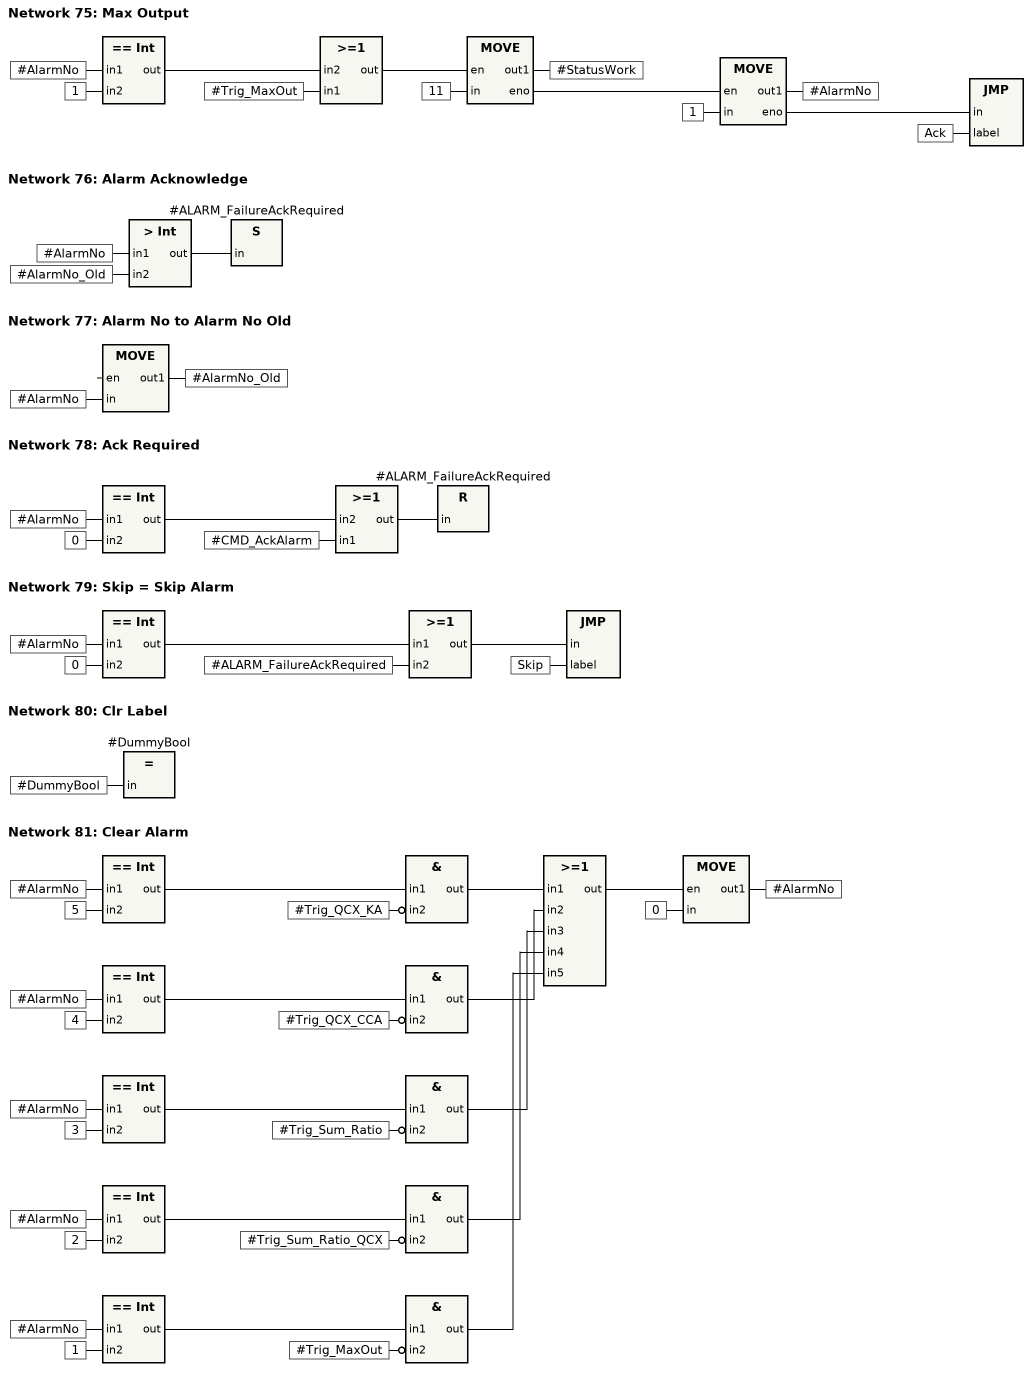
   // ENO of a box is taken as its EN; it also drops when the box reports an error
   #_w1 := (#AlarmNo = 1) OR #Trig_MaxOut;
   IF #_w1 THEN
       #StatusWork := 11;
       #AlarmNo := 1;
       GOTO Ack;
   END_IF;
END_REGION

REGION Network 76: Alarm Acknowledge
   Ack:
   IF #AlarmNo > #AlarmNo_Old THEN #ALARM_FailureAckRequired := TRUE; END_IF;
END_REGION

REGION Network 77: Alarm No to Alarm No Old
   #AlarmNo_Old := #AlarmNo;
END_REGION

REGION Network 78: Ack Required
   IF (#AlarmNo = 0) OR #CMD_AckAlarm THEN #ALARM_FailureAckRequired := FALSE; END_IF;
END_REGION

REGION Network 79: Skip = Skip Alarm
   IF (#AlarmNo = 0) OR #ALARM_FailureAckRequired THEN GOTO Skip; END_IF;
END_REGION

REGION Network 80: Clr Label
   Clr:
   #DummyBool := #DummyBool;
END_REGION

REGION Network 81: Clear Alarm
   IF ((#AlarmNo = 5) AND NOT #Trig_QCX_KA) OR ((#AlarmNo = 4) AND NOT #Trig_QCX_CCA) OR ((#AlarmNo = 3) AND NOT #Trig_Sum_Ratio) OR ((#AlarmNo = 2) AND NOT #Trig_Sum_Ratio_QCX) OR ((#AlarmNo = 1) AND NOT #Trig_MaxOut) THEN
       #AlarmNo := 0;
   END_IF;
END_REGION

REGION Network 82: Clear Alarm No Old
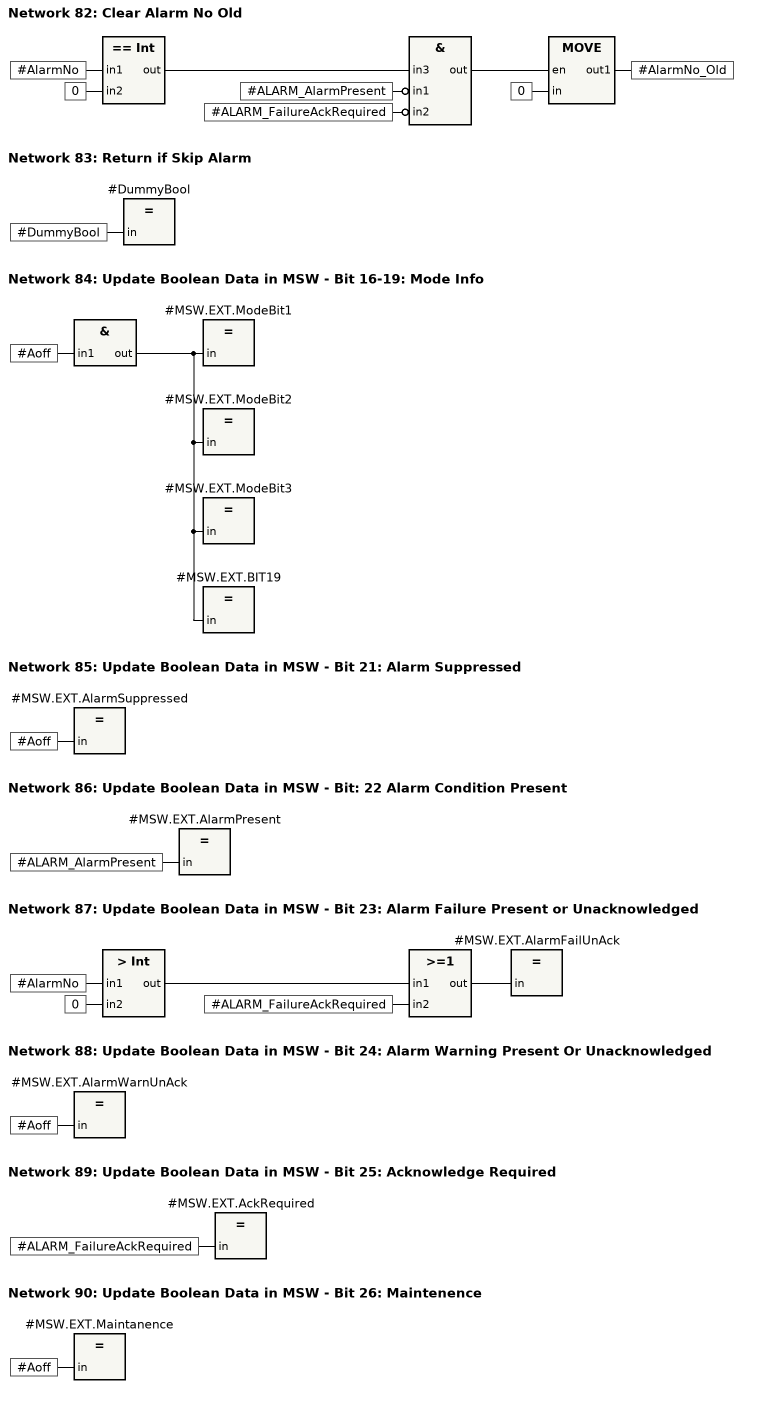
   IF (#AlarmNo = 0) AND NOT #ALARM_AlarmPresent AND NOT #ALARM_FailureAckRequired THEN
       #AlarmNo_Old := 0;
   END_IF;
END_REGION

REGION Network 83: Return if Skip Alarm
   Skip:
   #DummyBool := #DummyBool;
END_REGION

REGION Network 84: Update Boolean Data in MSW - Bit 16-19: Mode Info
   // 0 = Auto
   // 1= Single Start
   // 2 = Manual
   // 3= Local
   // 4= Test Mode
   #MSW.EXT.ModeBit1 := #Aoff;
   #MSW.EXT.ModeBit2 := #Aoff;
   #MSW.EXT.ModeBit3 := #Aoff;
   #MSW.EXT.BIT19 := #Aoff;
END_REGION

REGION Network 85: Update Boolean Data in MSW - Bit 21: Alarm Suppressed
   #MSW.EXT.AlarmSuppressed := #Aoff;
END_REGION

REGION Network 86: Update Boolean Data in MSW - Bit: 22 Alarm Condition Present
   #MSW.EXT.AlarmPresent := #ALARM_AlarmPresent;
END_REGION

REGION Network 87: Update Boolean Data in MSW - Bit 23: Alarm Failure Present or Unacknowledged
   #MSW.EXT.AlarmFailUnAck := (#AlarmNo > 0) OR #ALARM_FailureAckRequired;
END_REGION

REGION Network 88: Update Boolean Data in MSW - Bit 24: Alarm Warning Present Or Unacknowledged
   #MSW.EXT.AlarmWarnUnAck := #Aoff;
END_REGION

REGION Network 89: Update Boolean Data in MSW - Bit 25: Acknowledge Required
   #MSW.EXT.AckRequired := #ALARM_FailureAckRequired;
END_REGION

REGION Network 90: Update Boolean Data in MSW - Bit 26: Maintenence
   #MSW.EXT.Maintanence := #Aoff;
END_REGION

REGION Network 91: Update Boolean Data in MSW - Bit 27: Operation
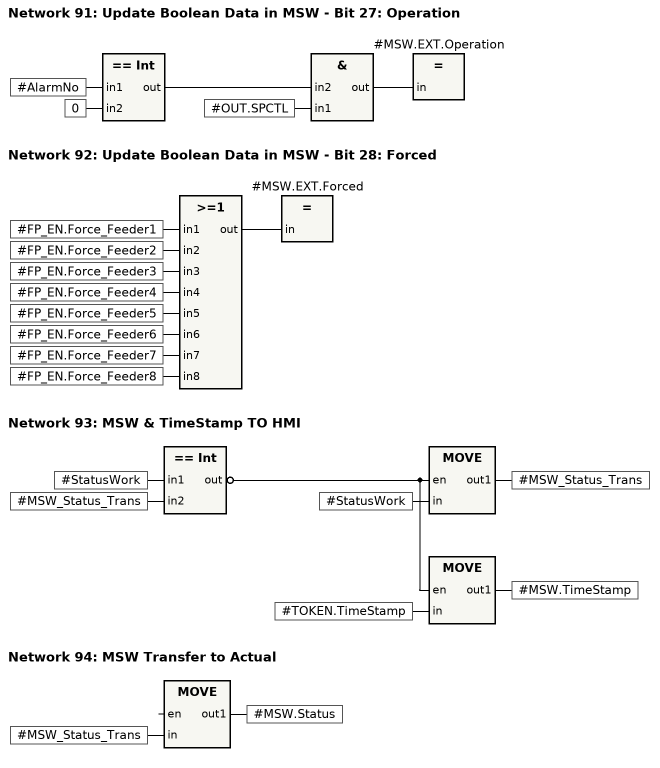
   #MSW.EXT.Operation := (#AlarmNo = 0) AND #OUT.SPCTL;
END_REGION

REGION Network 92: Update Boolean Data in MSW - Bit 28: Forced
   #MSW.EXT.Forced := #FP_EN.Force_Feeder1 OR #FP_EN.Force_Feeder2 OR #FP_EN.Force_Feeder3 OR #FP_EN.Force_Feeder4 OR #FP_EN.Force_Feeder5 OR #FP_EN.Force_Feeder6 OR #FP_EN.Force_Feeder7 OR #FP_EN.Force_Feeder8;
END_REGION

REGION Network 93: MSW & TimeStamp TO HMI
   #_w1 := NOT (#StatusWork = #MSW_Status_Trans);
   IF #_w1 THEN
       #MSW_Status_Trans := #StatusWork;
       #MSW.TimeStamp := #TOKEN.TimeStamp;
   END_IF;
END_REGION

REGION Network 94: MSW Transfer to Actual
   #MSW.Status := #MSW_Status_Trans;
END_REGION

REGION Network 95: Write STAT to OUT
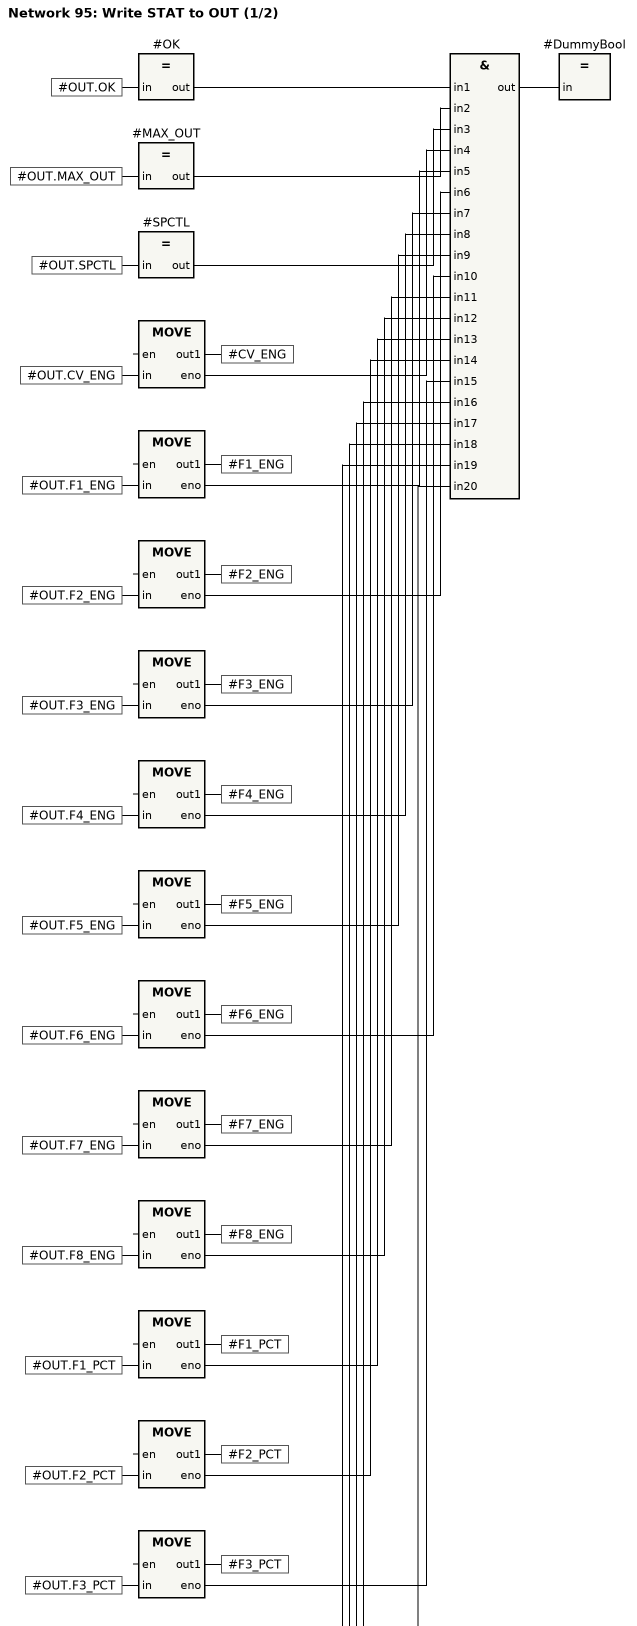
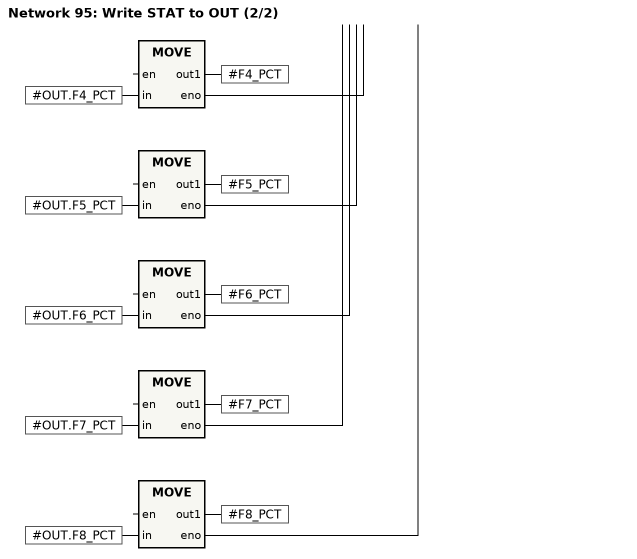
   #OK := #OUT.OK;
   #MAX_OUT := #OUT.MAX_OUT;
   #SPCTL := #OUT.SPCTL;
   #CV_ENG := #OUT.CV_ENG;
   #F1_ENG := #OUT.F1_ENG;
   #F2_ENG := #OUT.F2_ENG;
   #F3_ENG := #OUT.F3_ENG;
   #F4_ENG := #OUT.F4_ENG;
   #F5_ENG := #OUT.F5_ENG;
   #F6_ENG := #OUT.F6_ENG;
   #F7_ENG := #OUT.F7_ENG;
   #F8_ENG := #OUT.F8_ENG;
   #F1_PCT := #OUT.F1_PCT;
   #F2_PCT := #OUT.F2_PCT;
   #F3_PCT := #OUT.F3_PCT;
   #F4_PCT := #OUT.F4_PCT;
   #F5_PCT := #OUT.F5_PCT;
   #F6_PCT := #OUT.F6_PCT;
   #F7_PCT := #OUT.F7_PCT;
   #F8_PCT := #OUT.F8_PCT;
   #DummyBool := #OUT.OK AND #OUT.MAX_OUT AND #OUT.SPCTL;
END_REGION
END_FUNCTION_BLOCK

FUNCTION_BLOCK "ACESYS_SEQUENCE"   // FB231, FBD
TITLE = ACESYS V8.0 - Build 003 - SEQUENCE
{ S7_Optimized_Access := 'FALSE' }
AUTHOR : FLSmidth
FAMILY : ACESYS
NAME : SEQ
VERSION : 8.0
   VAR_INPUT
      TRANS_01 : Bool := TRUE;   // Transition 01
      TRANS_02 : Bool := TRUE;   // Transition 02
      TRANS_03 : Bool := TRUE;   // Transition 03
      TRANS_04 : Bool := TRUE;   // Transition 04
      TRANS_05 : Bool := TRUE;   // Transition 05
      TRANS_06 : Bool := TRUE;   // Transition 06
      TRANS_07 : Bool := TRUE;   // Transition 07
      TRANS_08 : Bool := TRUE;   // Transition 08
      TRANS_09 : Bool := TRUE;   // Transition 09
      TRANS_10 : Bool := TRUE;   // Transition 10
      TRANS_11 : Bool := TRUE;   // Transition 11
      TRANS_12 : Bool := TRUE;   // Transition 12
      TRANS_13 : Bool := TRUE;   // Transition 13
      TRANS_14 : Bool := TRUE;   // Transition 14
      TRANS_15 : Bool := TRUE;   // Transition 15
      TRANS_16 : Bool := TRUE;   // Transition 16
      RESET : Bool;   // Reset to Step 1
      SINGLE_STEP : Bool;   // Goto Next Step
      GOTO_STEP : Bool;   // Goto step Request
      GOTO_NO : Int;   // Goto step Number
   END_VAR
   VAR_OUTPUT
      OUT_01 : Bool;   // Output 01
      OUT_02 : Bool;   // Output 02
      OUT_03 : Bool;   // Output 03
      OUT_04 : Bool;   // Output 04
      OUT_05 : Bool;   // Output 05
      OUT_06 : Bool;   // Output 06
      OUT_07 : Bool;   // Output 07
      OUT_08 : Bool;   // Output 08
      OUT_09 : Bool;   // Output 09
      OUT_10 : Bool;   // Output 10
      OUT_11 : Bool;   // Output 11
      OUT_12 : Bool;   // Output 12
      OUT_13 : Bool;   // Output 13
      OUT_14 : Bool;   // Output 14
      OUT_15 : Bool;   // Output 15
      OUT_16 : Bool;   // Output 16
      OK : Bool := TRUE;   // Unit OK (1=no alarms)
      MAX_TIME : Bool;   // Max Step time exceeded
      ACT_STEP : Int;   // Actual Step
      MSW : "ACESYS_HMI_STAT_32T";
   END_VAR
   VAR_IN_OUT
      TOKEN : "ACESYS_TOKEN";
   END_VAR
   VAR
      BlockInfo : Struct
         Ace_Version : Int;   // Acesys Block Version Number
         Ace_BuildNo : Int;   // Acesys Block Build Number
         DB_Number : Int;   // Block Instance DB Number
      END_STRUCT;
      FP_CMD : Struct   // Faceplate Commands
         Spare_08 : Bool;
         Spare_09 : Bool;
         Spare_10 : Bool;
         Spare_11 : Bool;
         Spare_12 : Bool;
         Spare_13 : Bool;
         Spare_14 : Bool;
         AckAlarm : Bool;   // Alarm Acknowledge
         GotoStep1 : Bool;   // FacePlateCmd (bit 0): Reset Sequence to Step 1
         GotoNext : Bool;   // FacePlateCmd (bit 1): Goto Next STep
         Spare_02 : Bool;
         Spare_03 : Bool;
         Spare_04 : Bool;
         Spare_05 : Bool;
         Spare_06 : Bool;
         Spare_07 : Bool;
      END_STRUCT;
      FP_SEL : Struct
         Alarm_Type_1 : Bool;   // No Alarm
         Alarm_Type_2 : Bool;   // Alarm Warming
         Alarm_Type_3 : Bool;   // Alarm Failure
         Alarm_Type_4 : Bool;   // Spare (not Used)
         Alarm_Action_1 : Bool;   // No Action
         Alarm_Action_2 : Bool;   // Continue to next Step
         Alarm_Action_3 : Bool;   // Reset to Step 1
         Alarm_Action_4 : Bool;   // Spare (Not Used)
         Retentive_Timer : Bool;
      END_STRUCT;
      FP_PARM : Struct
         MATRIX : Array[1..16] of Word;   // Output Matrix
         Min_Time_Pre : Array[1..16] of DInt;   // Minumum Step Time
         Max_Time_Pre : Array[1..16] of DInt;   // Maximum Step Time
         Min_Time_Acc : DInt;   // Min Step time Actual
         Max_Time_Acc : DInt;   // Max Step time Actual
         Min_Time_SP : DInt;   // Min Step time Setpoint
         Max_Time_SP : DInt;   // Max Step time Setpoint
         NoOfOutputs : Int := 16;   // Number Outputs to be displayed on faceplate
         NoOfSteps : Int := 16;   // Number of Steps to be displayed on faceplate
         Min_Timer_EN : Bool;   // Minimum Step Timer Enabled
         Min_Timer_DN : Bool;   // Minimum Step Timer Elapsed
         Max_Timer_EN : Bool;   // Maximum Step Timer Enabled
         Max_Timer_DN : Bool;   // Maximum Step Time Elapsed
         Trans_Act : Bool;   // Active Transition
      END_STRUCT;
      FP_DIM : Struct
         GotoStep1 : Bool;
         GotoNext : Bool;
      END_STRUCT;
      FP_SHOW : Struct
         GotoStep1 : Bool;
         GotoNext : Bool;
      END_STRUCT;
      ONS : Struct
         Alarm_Type_1 : Bool;
         Alarm_Type_2 : Bool;
         Alarm_Type_3 : Bool;
         Alarm_Type_4 : Bool;
         Alarm_Action_1 : Bool;
         Alarm_Action_2 : Bool;
         Alarm_Action_3 : Bool;
         Alarm_Action_4 : Bool;
         Goto_Step : Bool;
         SingleStep : Bool;
         Reset : Bool;
         Acknowledge : Bool;
      END_STRUCT;
      Work_Step : Int;
      Old_Step : Int;
      StatusWork : Int;
      AlarmNo : Int;
      AlarmNo_Old : Int;
      TimerMin_SP : DInt;
      TimerMin_ACC : DInt;
      TimerMax_SP : DInt;
      TimerMax_ACC : DInt;
      Reset_Timer : Bool;
      ALARM_AlarmPresent : Bool;
      ALARM_WarnPresent : Bool;
      ALARM_FailureAckRequired : Bool;
      ALARM_Warn_Ack_Required : Bool;
      CMD_Acknowledge : Bool;
      Min_Timer : TONR_TIME;
      Max_Timer : TONR_TIME;
      MSW_Status_Trans : Int;
      OUT : Struct
         OUT_01 : Bool;
         OUT_02 : Bool;
         OUT_03 : Bool;
         OUT_04 : Bool;
         OUT_05 : Bool;
         OUT_06 : Bool;
         OUT_07 : Bool;
         OUT_08 : Bool;
         OUT_09 : Bool;
         OUT_10 : Bool;
         OUT_11 : Bool;
         OUT_12 : Bool;
         OUT_13 : Bool;
         OUT_14 : Bool;
         OUT_15 : Bool;
         OUT_16 : Bool;
         OK : Bool;
         MAX_TIME : Bool;
      END_STRUCT;
      Min_Timer_Q : Bool;
      Max_Timer_Q : Bool;
   END_VAR
   VAR_TEMP
      Aon : Bool;
      Aoff : Bool;
      DummyBool : Bool;
      Work_Matrix : Word;
      Work_Matrix_B AT Work_Matrix : Array[0..15] of Bool;
   END_VAR
   VAR_TEMP   // added for the SCL form of the ladder/FBD networks
      _w1 : Bool;
      _w2 : Bool;
      _w3 : Bool;
      _w4 : Bool;
      _w5 : Bool;
      _w6 : Bool;
      _w7 : Bool;
      _w8 : Bool;
      _w9 : Bool;
      _w10 : Bool;
      _w11 : Bool;
      _w12 : Bool;
      _w13 : Bool;
      _w14 : Bool;
      _w15 : Bool;
      _w16 : Bool;
   END_VAR
BEGIN

REGION Network 1
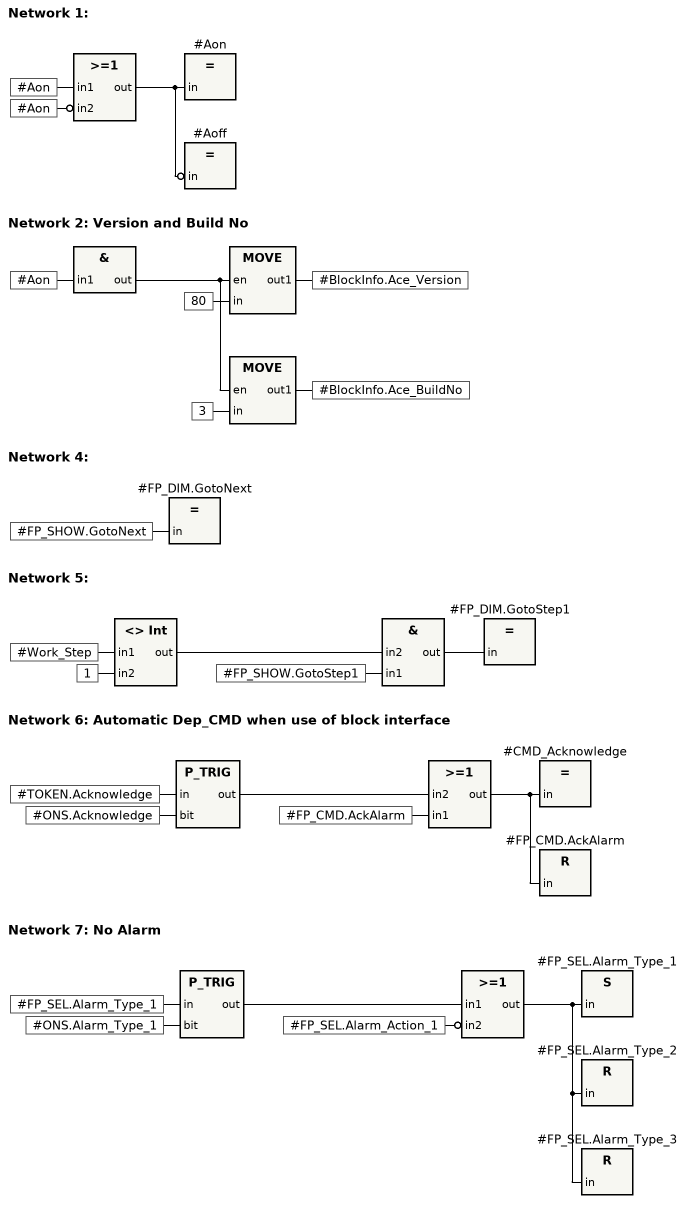
   #Aon := #Aon OR NOT #Aon;
   #Aoff := NOT #Aon;
END_REGION

REGION Network 2: Version and Build No
   IF #Aon THEN
       #BlockInfo.Ace_Version := 80;
       #BlockInfo.Ace_BuildNo := 3;
   END_IF;
END_REGION

REGION Network 3 (STL): Instance DB Number to Faceplate
         L     DINO;
         T     #BlockInfo.DB_Number;
END_REGION

REGION Network 4
   #FP_DIM.GotoNext := #FP_SHOW.GotoNext;
END_REGION

REGION Network 5
   #FP_DIM.GotoStep1 := (#Work_Step <> 1) AND #FP_SHOW.GotoStep1;
END_REGION

REGION Network 6: Automatic Dep_CMD when use of block interface
   #_w1 := #TOKEN.Acknowledge AND NOT #ONS.Acknowledge;   // rising edge
   #ONS.Acknowledge := #TOKEN.Acknowledge;
   #CMD_Acknowledge := #_w1 OR #FP_CMD.AckAlarm;
   IF #CMD_Acknowledge THEN #FP_CMD.AckAlarm := FALSE; END_IF;
END_REGION

REGION Network 7: No Alarm
   // Alarm Type:
   // 
   // 1 = No Alarm
   // 2 = Alarm Warning
   // 3 = Alarm Failure
   #_w1 := #FP_SEL.Alarm_Type_1 AND NOT #ONS.Alarm_Type_1;   // rising edge
   #ONS.Alarm_Type_1 := #FP_SEL.Alarm_Type_1;
   IF #_w1 OR NOT #FP_SEL.Alarm_Action_1 THEN
       #FP_SEL.Alarm_Type_1 := TRUE;
       #FP_SEL.Alarm_Type_2 := FALSE;
       #FP_SEL.Alarm_Type_3 := FALSE;
   END_IF;
END_REGION

REGION Network 8: No Alarm
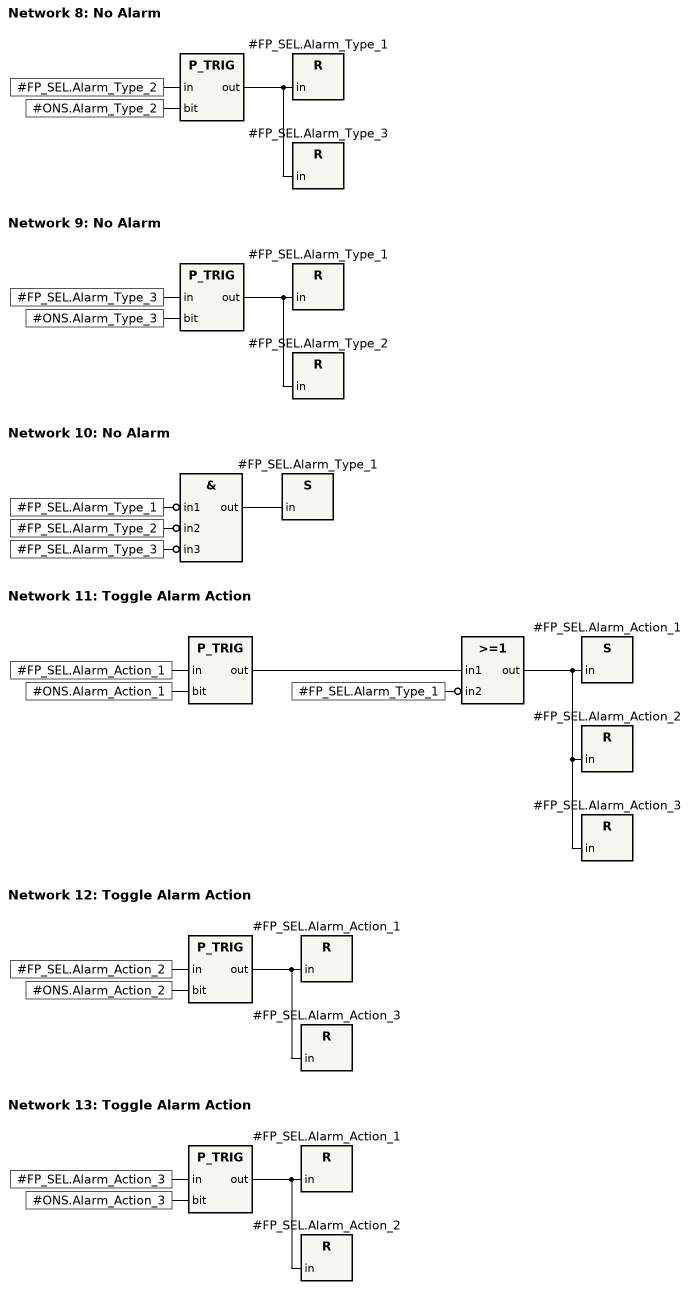
   #_w1 := #FP_SEL.Alarm_Type_2 AND NOT #ONS.Alarm_Type_2;   // rising edge
   #ONS.Alarm_Type_2 := #FP_SEL.Alarm_Type_2;
   IF #_w1 THEN
       #FP_SEL.Alarm_Type_1 := FALSE;
       #FP_SEL.Alarm_Type_3 := FALSE;
   END_IF;
END_REGION

REGION Network 9: No Alarm
   #_w1 := #FP_SEL.Alarm_Type_3 AND NOT #ONS.Alarm_Type_3;   // rising edge
   #ONS.Alarm_Type_3 := #FP_SEL.Alarm_Type_3;
   IF #_w1 THEN
       #FP_SEL.Alarm_Type_1 := FALSE;
       #FP_SEL.Alarm_Type_2 := FALSE;
   END_IF;
END_REGION

REGION Network 10: No Alarm
   IF NOT #FP_SEL.Alarm_Type_1 AND NOT #FP_SEL.Alarm_Type_2 AND NOT #FP_SEL.Alarm_Type_3 THEN
       #FP_SEL.Alarm_Type_1 := TRUE;
   END_IF;
END_REGION

REGION Network 11: Toggle Alarm Action
   // Alarm Action:
   // 
   // 1 = No Action
   // 2 = Continue to Next Step
   // 3 = Reset to Step 1
   // 4 = Stay in current step until Alarm Acknowledged
   #_w1 := #FP_SEL.Alarm_Action_1 AND NOT #ONS.Alarm_Action_1;   // rising edge
   #ONS.Alarm_Action_1 := #FP_SEL.Alarm_Action_1;
   IF #_w1 OR NOT #FP_SEL.Alarm_Type_1 THEN
       #FP_SEL.Alarm_Action_1 := TRUE;
       #FP_SEL.Alarm_Action_2 := FALSE;
       #FP_SEL.Alarm_Action_3 := FALSE;
   END_IF;
END_REGION

REGION Network 12: Toggle Alarm Action
   #_w1 := #FP_SEL.Alarm_Action_2 AND NOT #ONS.Alarm_Action_2;   // rising edge
   #ONS.Alarm_Action_2 := #FP_SEL.Alarm_Action_2;
   IF #_w1 THEN
       #FP_SEL.Alarm_Action_1 := FALSE;
       #FP_SEL.Alarm_Action_3 := FALSE;
   END_IF;
END_REGION

REGION Network 13: Toggle Alarm Action
   #_w1 := #FP_SEL.Alarm_Action_3 AND NOT #ONS.Alarm_Action_3;   // rising edge
   #ONS.Alarm_Action_3 := #FP_SEL.Alarm_Action_3;
   IF #_w1 THEN
       #FP_SEL.Alarm_Action_1 := FALSE;
       #FP_SEL.Alarm_Action_2 := FALSE;
   END_IF;
END_REGION

REGION Network 14: No Action
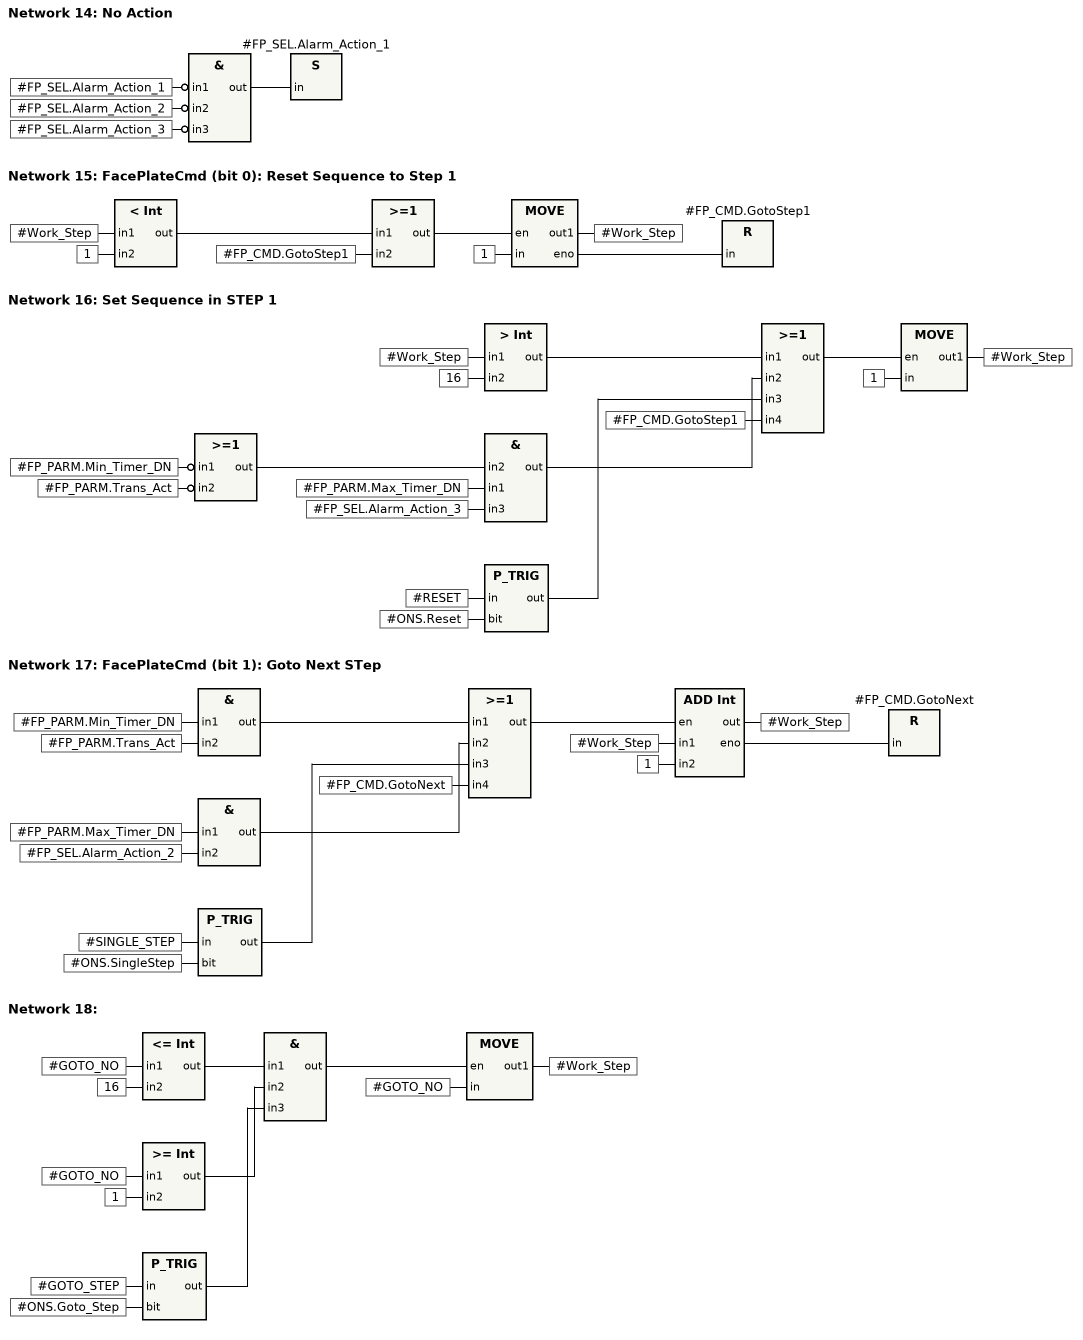
   IF NOT #FP_SEL.Alarm_Action_1 AND NOT #FP_SEL.Alarm_Action_2 AND NOT #FP_SEL.Alarm_Action_3 THEN
       #FP_SEL.Alarm_Action_1 := TRUE;
   END_IF;
END_REGION

REGION Network 15: FacePlateCmd (bit 0): Reset Sequence to Step 1
   // ENO of a box is taken as its EN; it also drops when the box reports an error
   #_w1 := (#Work_Step < 1) OR #FP_CMD.GotoStep1;
   IF #_w1 THEN
       #Work_Step := 1;
       #FP_CMD.GotoStep1 := FALSE;
   END_IF;
END_REGION

REGION Network 16: Set Sequence in STEP 1
   #_w1 := #RESET AND NOT #ONS.Reset;   // rising edge
   #ONS.Reset := #RESET;
   IF (#Work_Step > 16) OR ((NOT #FP_PARM.Min_Timer_DN OR NOT #FP_PARM.Trans_Act) AND #FP_PARM.Max_Timer_DN AND #FP_SEL.Alarm_Action_3) OR #_w1 OR #FP_CMD.GotoStep1 THEN
       #Work_Step := 1;
   END_IF;
END_REGION

REGION Network 17: FacePlateCmd (bit 1): Goto Next STep
   // ENO of a box is taken as its EN; it also drops when the box reports an error
   #_w1 := #SINGLE_STEP AND NOT #ONS.SingleStep;   // rising edge
   #ONS.SingleStep := #SINGLE_STEP;
   IF (#FP_PARM.Min_Timer_DN AND #FP_PARM.Trans_Act) OR (#FP_PARM.Max_Timer_DN AND #FP_SEL.Alarm_Action_2) OR #_w1 OR #FP_CMD.GotoNext THEN
       #Work_Step := #Work_Step + 1;
       #FP_CMD.GotoNext := FALSE;
   END_IF;
END_REGION

REGION Network 18
   #_w1 := #GOTO_STEP AND NOT #ONS.Goto_Step;   // rising edge
   #ONS.Goto_Step := #GOTO_STEP;
   IF (#GOTO_NO <= 16) AND (#GOTO_NO >= 1) AND #_w1 THEN #Work_Step := #GOTO_NO; END_IF;
END_REGION

REGION Network 19
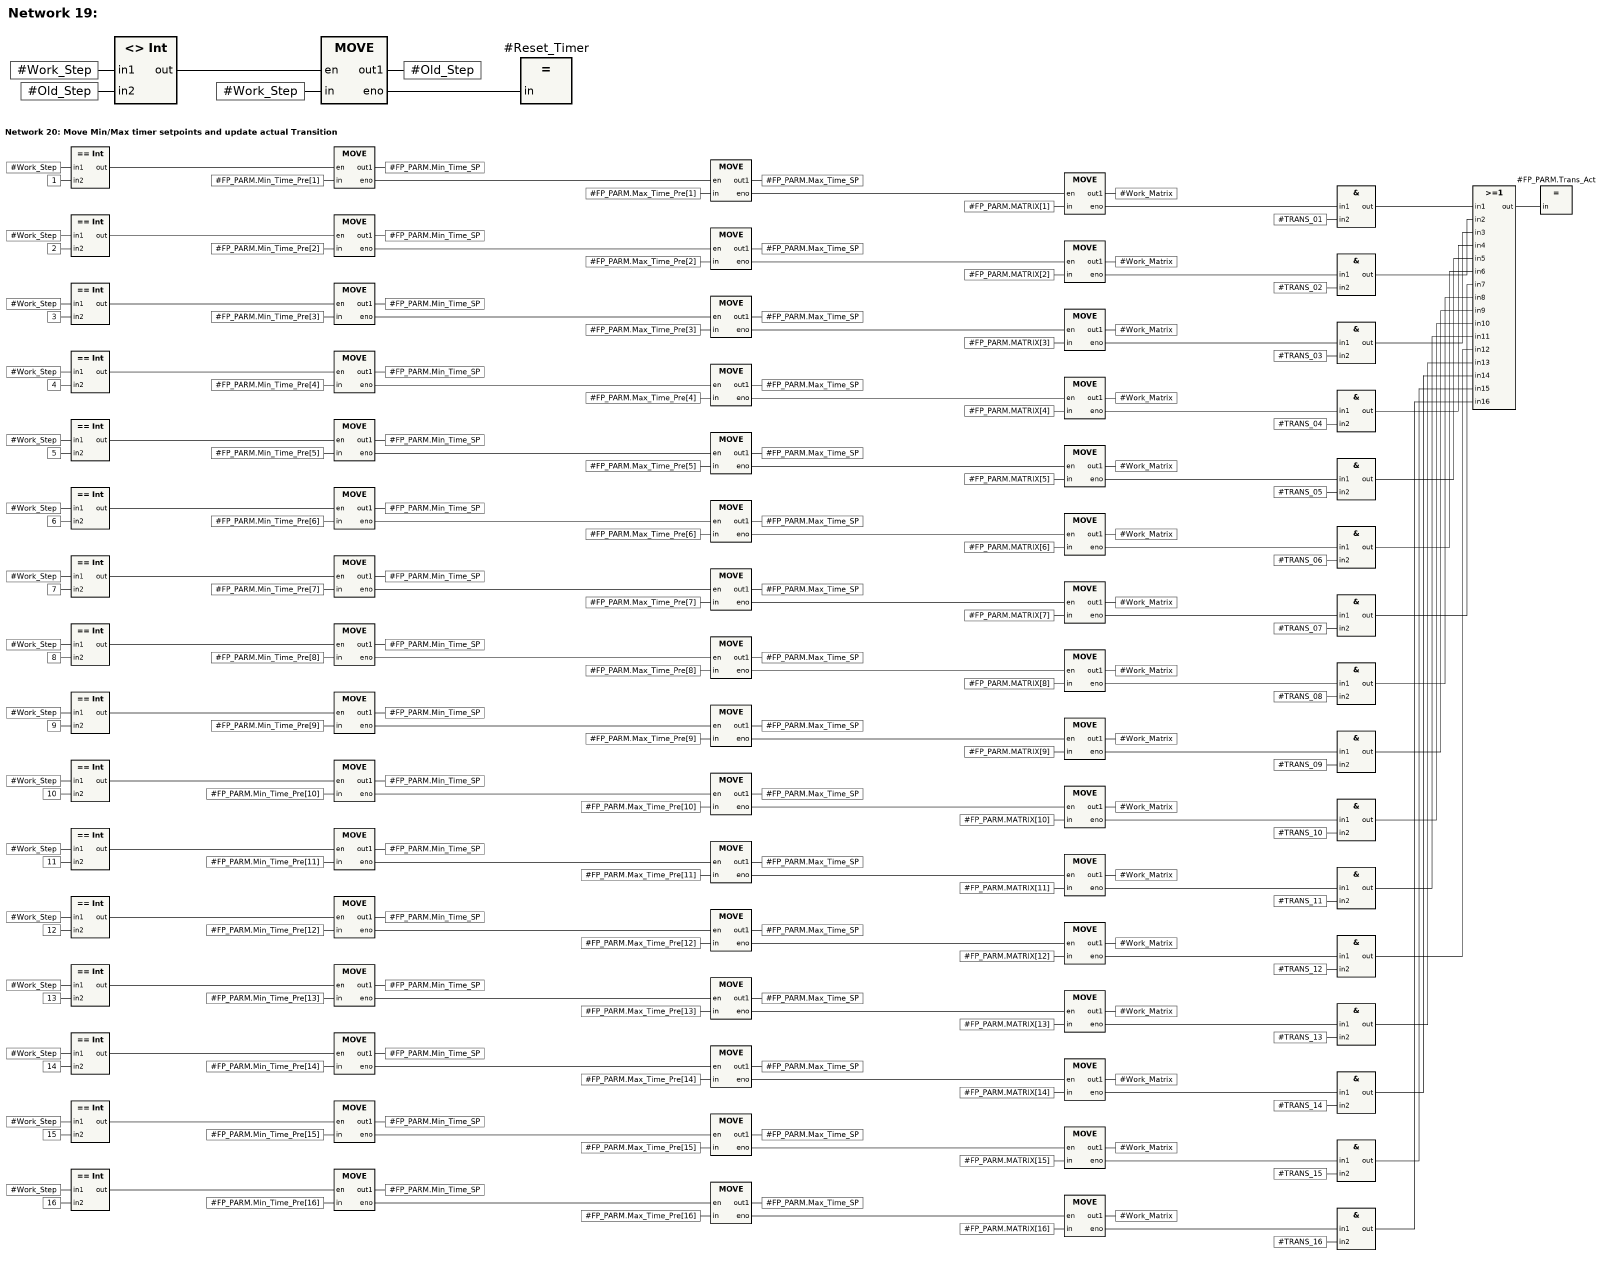
   // ENO of a box is taken as its EN; it also drops when the box reports an error
   #_w1 := #Work_Step <> #Old_Step;
   IF #_w1 THEN #Old_Step := #Work_Step; END_IF;
   #Reset_Timer := #_w1;
END_REGION

REGION Network 20: Move Min/Max timer setpoints and update actual Transition
   // ENO of a box is taken as its EN; it also drops when the box reports an error
   #_w1 := #Work_Step = 1;
   IF #_w1 THEN
       #FP_PARM.Min_Time_SP := #FP_PARM.Min_Time_Pre[1];
       #FP_PARM.Max_Time_SP := #FP_PARM.Max_Time_Pre[1];
       #Work_Matrix := #FP_PARM.MATRIX[1];
   END_IF;
   #_w2 := #Work_Step = 2;
   IF #_w2 THEN
       #FP_PARM.Min_Time_SP := #FP_PARM.Min_Time_Pre[2];
       #FP_PARM.Max_Time_SP := #FP_PARM.Max_Time_Pre[2];
       #Work_Matrix := #FP_PARM.MATRIX[2];
   END_IF;
   #_w3 := #Work_Step = 3;
   IF #_w3 THEN
       #FP_PARM.Min_Time_SP := #FP_PARM.Min_Time_Pre[3];
       #FP_PARM.Max_Time_SP := #FP_PARM.Max_Time_Pre[3];
       #Work_Matrix := #FP_PARM.MATRIX[3];
   END_IF;
   #_w4 := #Work_Step = 4;
   IF #_w4 THEN
       #FP_PARM.Min_Time_SP := #FP_PARM.Min_Time_Pre[4];
       #FP_PARM.Max_Time_SP := #FP_PARM.Max_Time_Pre[4];
       #Work_Matrix := #FP_PARM.MATRIX[4];
   END_IF;
   #_w5 := #Work_Step = 5;
   IF #_w5 THEN
       #FP_PARM.Min_Time_SP := #FP_PARM.Min_Time_Pre[5];
       #FP_PARM.Max_Time_SP := #FP_PARM.Max_Time_Pre[5];
       #Work_Matrix := #FP_PARM.MATRIX[5];
   END_IF;
   #_w6 := #Work_Step = 6;
   IF #_w6 THEN
       #FP_PARM.Min_Time_SP := #FP_PARM.Min_Time_Pre[6];
       #FP_PARM.Max_Time_SP := #FP_PARM.Max_Time_Pre[6];
       #Work_Matrix := #FP_PARM.MATRIX[6];
   END_IF;
   #_w7 := #Work_Step = 7;
   IF #_w7 THEN
       #FP_PARM.Min_Time_SP := #FP_PARM.Min_Time_Pre[7];
       #FP_PARM.Max_Time_SP := #FP_PARM.Max_Time_Pre[7];
       #Work_Matrix := #FP_PARM.MATRIX[7];
   END_IF;
   #_w8 := #Work_Step = 8;
   IF #_w8 THEN
       #FP_PARM.Min_Time_SP := #FP_PARM.Min_Time_Pre[8];
       #FP_PARM.Max_Time_SP := #FP_PARM.Max_Time_Pre[8];
       #Work_Matrix := #FP_PARM.MATRIX[8];
   END_IF;
   #_w9 := #Work_Step = 9;
   IF #_w9 THEN
       #FP_PARM.Min_Time_SP := #FP_PARM.Min_Time_Pre[9];
       #FP_PARM.Max_Time_SP := #FP_PARM.Max_Time_Pre[9];
       #Work_Matrix := #FP_PARM.MATRIX[9];
   END_IF;
   #_w10 := #Work_Step = 10;
   IF #_w10 THEN
       #FP_PARM.Min_Time_SP := #FP_PARM.Min_Time_Pre[10];
       #FP_PARM.Max_Time_SP := #FP_PARM.Max_Time_Pre[10];
       #Work_Matrix := #FP_PARM.MATRIX[10];
   END_IF;
   #_w11 := #Work_Step = 11;
   IF #_w11 THEN
       #FP_PARM.Min_Time_SP := #FP_PARM.Min_Time_Pre[11];
       #FP_PARM.Max_Time_SP := #FP_PARM.Max_Time_Pre[11];
       #Work_Matrix := #FP_PARM.MATRIX[11];
   END_IF;
   #_w12 := #Work_Step = 12;
   IF #_w12 THEN
       #FP_PARM.Min_Time_SP := #FP_PARM.Min_Time_Pre[12];
       #FP_PARM.Max_Time_SP := #FP_PARM.Max_Time_Pre[12];
       #Work_Matrix := #FP_PARM.MATRIX[12];
   END_IF;
   #_w13 := #Work_Step = 13;
   IF #_w13 THEN
       #FP_PARM.Min_Time_SP := #FP_PARM.Min_Time_Pre[13];
       #FP_PARM.Max_Time_SP := #FP_PARM.Max_Time_Pre[13];
       #Work_Matrix := #FP_PARM.MATRIX[13];
   END_IF;
   #_w14 := #Work_Step = 14;
   IF #_w14 THEN
       #FP_PARM.Min_Time_SP := #FP_PARM.Min_Time_Pre[14];
       #FP_PARM.Max_Time_SP := #FP_PARM.Max_Time_Pre[14];
       #Work_Matrix := #FP_PARM.MATRIX[14];
   END_IF;
   #_w15 := #Work_Step = 15;
   IF #_w15 THEN
       #FP_PARM.Min_Time_SP := #FP_PARM.Min_Time_Pre[15];
       #FP_PARM.Max_Time_SP := #FP_PARM.Max_Time_Pre[15];
       #Work_Matrix := #FP_PARM.MATRIX[15];
   END_IF;
   #_w16 := #Work_Step = 16;
   IF #_w16 THEN
       #FP_PARM.Min_Time_SP := #FP_PARM.Min_Time_Pre[16];
       #FP_PARM.Max_Time_SP := #FP_PARM.Max_Time_Pre[16];
       #Work_Matrix := #FP_PARM.MATRIX[16];
   END_IF;
   #FP_PARM.Trans_Act := (#_w1 AND #TRANS_01) OR (#_w2 AND #TRANS_02) OR (#_w3 AND #TRANS_03) OR (#_w4 AND #TRANS_04) OR (#_w5 AND #TRANS_05) OR (#_w6 AND #TRANS_06) OR (#_w7 AND #TRANS_07) OR (#_w8 AND #TRANS_08) OR (#_w9 AND #TRANS_09) OR (#_w10 AND #TRANS_10) OR (#_w11 AND #TRANS_11) OR (#_w12 AND #TRANS_12) OR (#_w13 AND #TRANS_13) OR (#_w14 AND #TRANS_14) OR (#_w15 AND #TRANS_15) OR (#_w16 AND #TRANS_16);
END_REGION

REGION Network 21: Convert from 1/10 sec to mili sec.
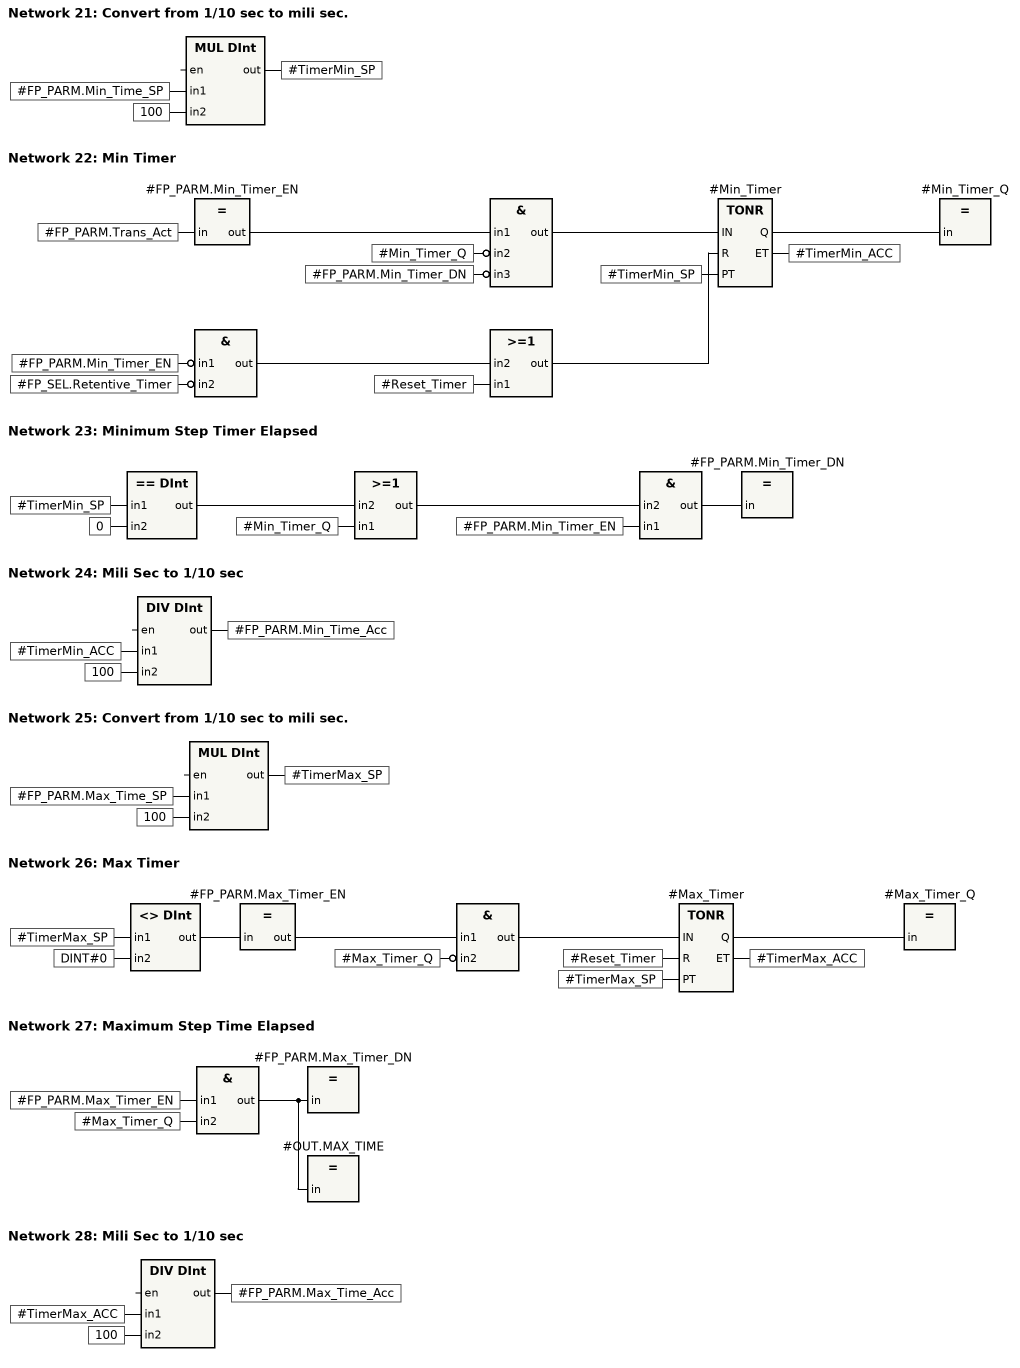
   #TimerMin_SP := #FP_PARM.Min_Time_SP * 100;
END_REGION

REGION Network 22: Min Timer
   // Build 003 - 05. May 2020 (EXTBOB) : Min_Timer_Q output created and used in place Min_Timer.Q
   #FP_PARM.Min_Timer_EN := #FP_PARM.Trans_Act;
   #Min_Timer(IN := #FP_PARM.Trans_Act AND NOT #Min_Timer_Q AND NOT #FP_PARM.Min_Timer_DN,   // TONR
              R := (NOT #FP_PARM.Min_Timer_EN AND NOT #FP_SEL.Retentive_Timer) OR #Reset_Timer,
              PT := #TimerMin_SP,
              ET => #TimerMin_ACC);
   #Min_Timer_Q := #Min_Timer.Q;
END_REGION

REGION Network 23: Minimum Step Timer Elapsed
   // Build 002 - 30. Jul 2019 (EXTBOB) : If minimum timer SP = 0 then move to next step added
   // Build 003 - 05. May 2020 (EXTBOB) : Min_Timer_Q used in place Min_Timer.Q
   #FP_PARM.Min_Timer_DN := ((#TimerMin_SP = 0) OR #Min_Timer_Q) AND #FP_PARM.Min_Timer_EN;
END_REGION

REGION Network 24: Mili Sec to 1/10 sec
   #FP_PARM.Min_Time_Acc := #TimerMin_ACC / 100;
END_REGION

REGION Network 25: Convert from 1/10 sec to mili sec.
   #TimerMax_SP := #FP_PARM.Max_Time_SP * 100;
END_REGION

REGION Network 26: Max Timer
   // Build 003 - 05. May 2020 (EXTBOB) : Max_Timer_Q output created and used in place Max_Timer.Q
   #FP_PARM.Max_Timer_EN := #TimerMax_SP <> DINT#0;
   #Max_Timer(IN := #FP_PARM.Max_Timer_EN AND NOT #Max_Timer_Q,   // TONR
              R := #Reset_Timer,
              PT := #TimerMax_SP,
              ET => #TimerMax_ACC);
   #Max_Timer_Q := #Max_Timer.Q;
END_REGION

REGION Network 27: Maximum Step Time Elapsed
   // Build 003 - 05. May 2020 (EXTBOB) : Max_Timer_Q output used in place Max_Timer.Q
   #FP_PARM.Max_Timer_DN := #FP_PARM.Max_Timer_EN AND #Max_Timer_Q;
   #OUT.MAX_TIME := #FP_PARM.Max_Timer_DN;
END_REGION

REGION Network 28: Mili Sec to 1/10 sec
   #FP_PARM.Max_Time_Acc := #TimerMax_ACC / 100;
END_REGION

REGION Network 29
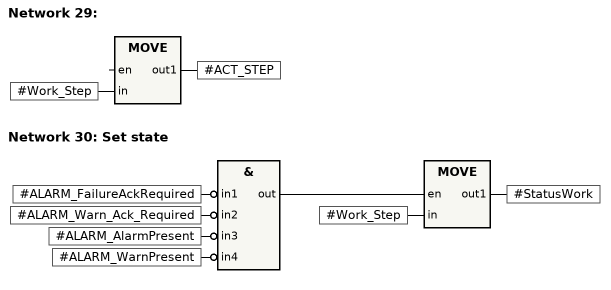
   #ACT_STEP := #Work_Step;
END_REGION

REGION Network 30: Set state
   IF NOT #ALARM_FailureAckRequired AND NOT #ALARM_Warn_Ack_Required AND NOT #ALARM_AlarmPresent AND NOT #ALARM_WarnPresent THEN
       #StatusWork := #Work_Step;
   END_IF;
END_REGION

REGION Network 31: Output
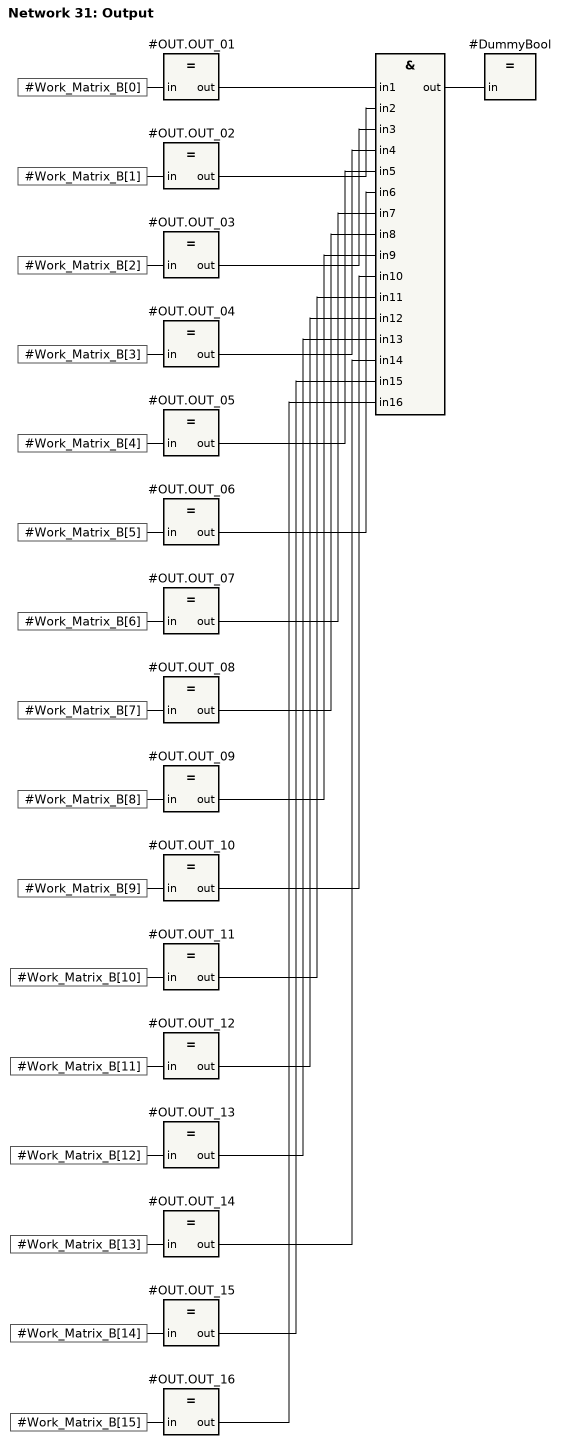
   #OUT.OUT_01 := #Work_Matrix_B[0];
   #OUT.OUT_02 := #Work_Matrix_B[1];
   #OUT.OUT_03 := #Work_Matrix_B[2];
   #OUT.OUT_04 := #Work_Matrix_B[3];
   #OUT.OUT_05 := #Work_Matrix_B[4];
   #OUT.OUT_06 := #Work_Matrix_B[5];
   #OUT.OUT_07 := #Work_Matrix_B[6];
   #OUT.OUT_08 := #Work_Matrix_B[7];
   #OUT.OUT_09 := #Work_Matrix_B[8];
   #OUT.OUT_10 := #Work_Matrix_B[9];
   #OUT.OUT_11 := #Work_Matrix_B[10];
   #OUT.OUT_12 := #Work_Matrix_B[11];
   #OUT.OUT_13 := #Work_Matrix_B[12];
   #OUT.OUT_14 := #Work_Matrix_B[13];
   #OUT.OUT_15 := #Work_Matrix_B[14];
   #OUT.OUT_16 := #Work_Matrix_B[15];
   #DummyBool := #Work_Matrix_B[0] AND #Work_Matrix_B[1] AND #Work_Matrix_B[2] AND #Work_Matrix_B[3] AND #Work_Matrix_B[4] AND #Work_Matrix_B[5] AND #Work_Matrix_B[6] AND #Work_Matrix_B[7] AND #Work_Matrix_B[8] AND #Work_Matrix_B[9] AND #Work_Matrix_B[10] AND #Work_Matrix_B[11] AND #Work_Matrix_B[12] AND #Work_Matrix_B[13] AND #Work_Matrix_B[14] AND #Work_Matrix_B[15];
END_REGION

REGION Network 32: Unit OK (1=no alarms)
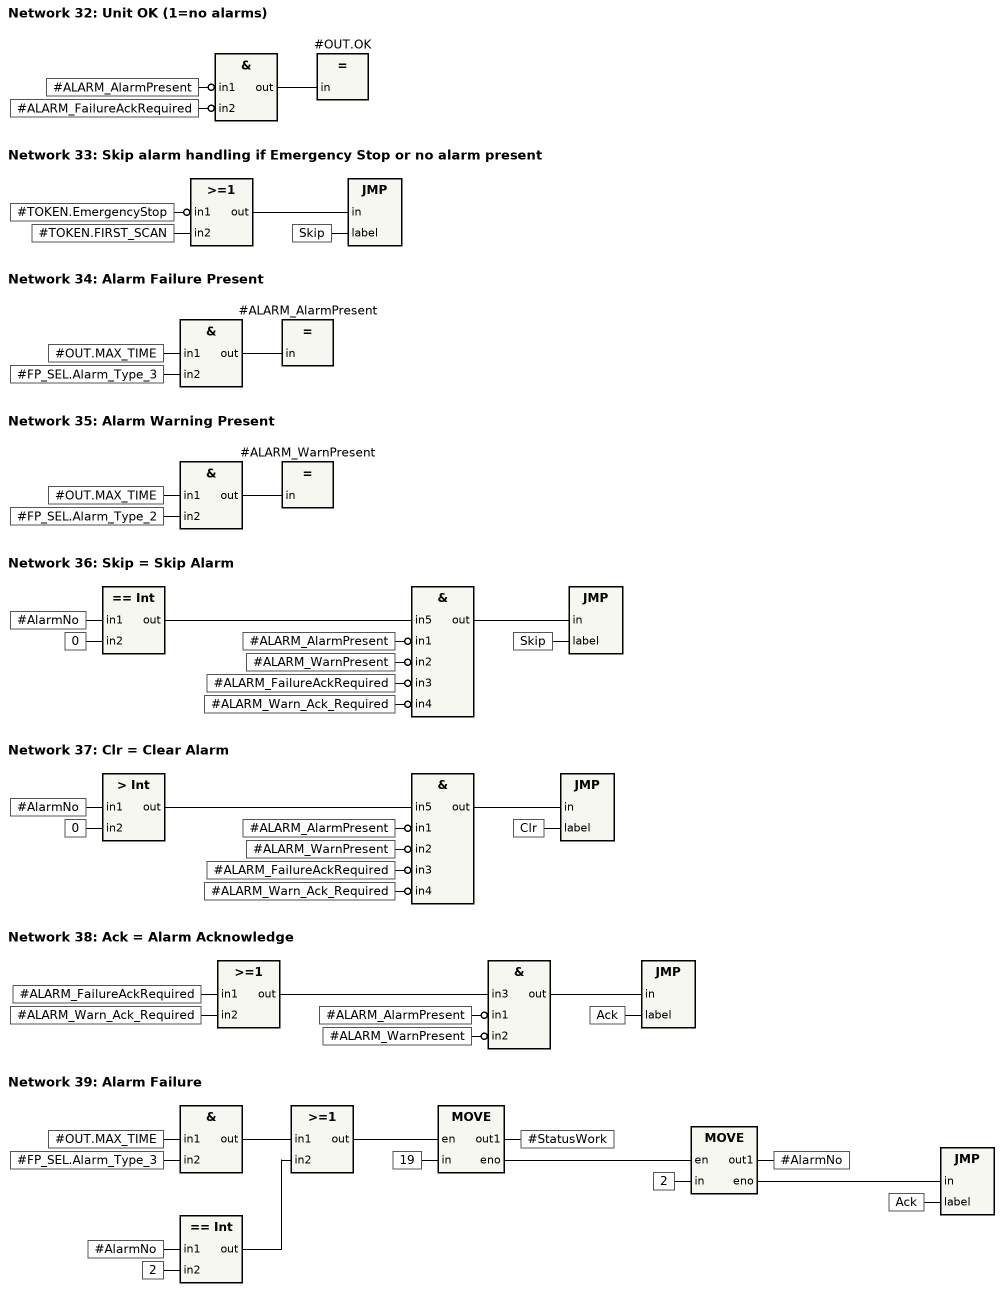
   #OUT.OK := NOT #ALARM_AlarmPresent AND NOT #ALARM_FailureAckRequired;
END_REGION

REGION Network 33: Skip alarm handling if Emergency Stop or no alarm present
   // Skip = Skip Alarm
   IF NOT #TOKEN.EmergencyStop OR #TOKEN.FIRST_SCAN THEN GOTO Skip; END_IF;
END_REGION

REGION Network 34: Alarm Failure Present
   #ALARM_AlarmPresent := #OUT.MAX_TIME AND #FP_SEL.Alarm_Type_3;
END_REGION

REGION Network 35: Alarm Warning Present
   #ALARM_WarnPresent := #OUT.MAX_TIME AND #FP_SEL.Alarm_Type_2;
END_REGION

REGION Network 36: Skip = Skip Alarm
   IF (#AlarmNo = 0) AND NOT #ALARM_AlarmPresent AND NOT #ALARM_WarnPresent AND NOT #ALARM_FailureAckRequired AND NOT #ALARM_Warn_Ack_Required THEN
       GOTO Skip;
   END_IF;
END_REGION

REGION Network 37: Clr = Clear Alarm
   IF (#AlarmNo > 0) AND NOT #ALARM_AlarmPresent AND NOT #ALARM_WarnPresent AND NOT #ALARM_FailureAckRequired AND NOT #ALARM_Warn_Ack_Required THEN
       GOTO Clr;
   END_IF;
END_REGION

REGION Network 38: Ack = Alarm Acknowledge
   IF (#ALARM_FailureAckRequired OR #ALARM_Warn_Ack_Required) AND NOT #ALARM_AlarmPresent AND NOT #ALARM_WarnPresent THEN
       GOTO Ack;
   END_IF;
END_REGION

REGION Network 39: Alarm Failure
   // ENO of a box is taken as its EN; it also drops when the box reports an error
   #_w1 := (#OUT.MAX_TIME AND #FP_SEL.Alarm_Type_3) OR (#AlarmNo = 2);
   IF #_w1 THEN
       #StatusWork := 19;
       #AlarmNo := 2;
       GOTO Ack;
   END_IF;
END_REGION

REGION Network 40: Alarm Warning
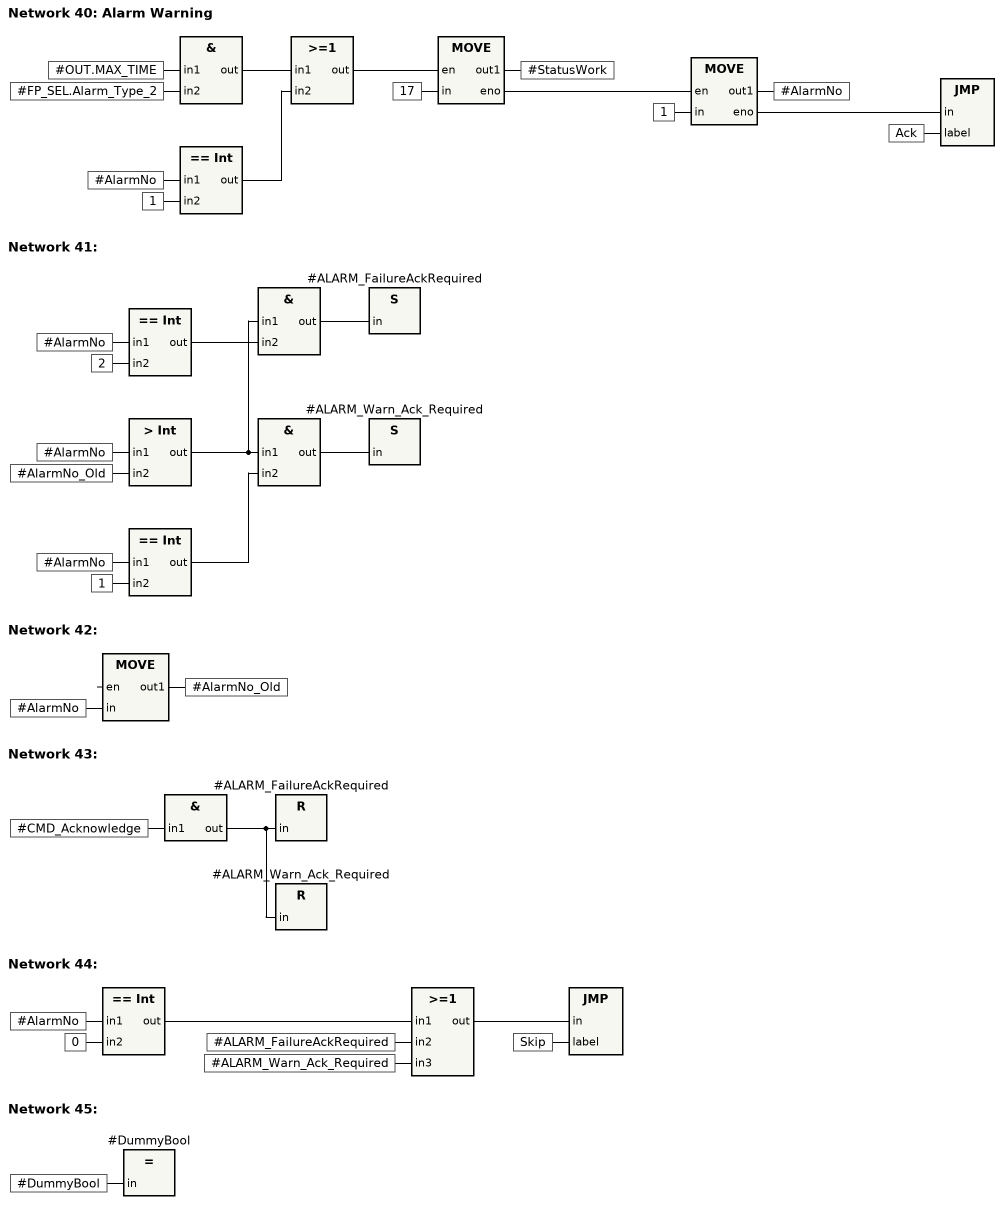
   // ENO of a box is taken as its EN; it also drops when the box reports an error
   #_w1 := (#OUT.MAX_TIME AND #FP_SEL.Alarm_Type_2) OR (#AlarmNo = 1);
   IF #_w1 THEN
       #StatusWork := 17;
       #AlarmNo := 1;
       GOTO Ack;
   END_IF;
END_REGION

REGION Network 41
   // ***Alarm Acknowledge***
   Ack:
   #_w1 := #AlarmNo > #AlarmNo_Old;
   IF #_w1 AND (#AlarmNo = 2) THEN #ALARM_FailureAckRequired := TRUE; END_IF;
   IF #_w1 AND (#AlarmNo = 1) THEN #ALARM_Warn_Ack_Required := TRUE; END_IF;
END_REGION

REGION Network 42
   #AlarmNo_Old := #AlarmNo;
END_REGION

REGION Network 43
   IF #CMD_Acknowledge THEN
       #ALARM_FailureAckRequired := FALSE;
       #ALARM_Warn_Ack_Required := FALSE;
   END_IF;
END_REGION

REGION Network 44
   // Skip = Skip Alarm
   IF (#AlarmNo = 0) OR #ALARM_FailureAckRequired OR #ALARM_Warn_Ack_Required THEN GOTO Skip; END_IF;
END_REGION

REGION Network 45
   Clr:
   #DummyBool := #DummyBool;
END_REGION

REGION Network 46
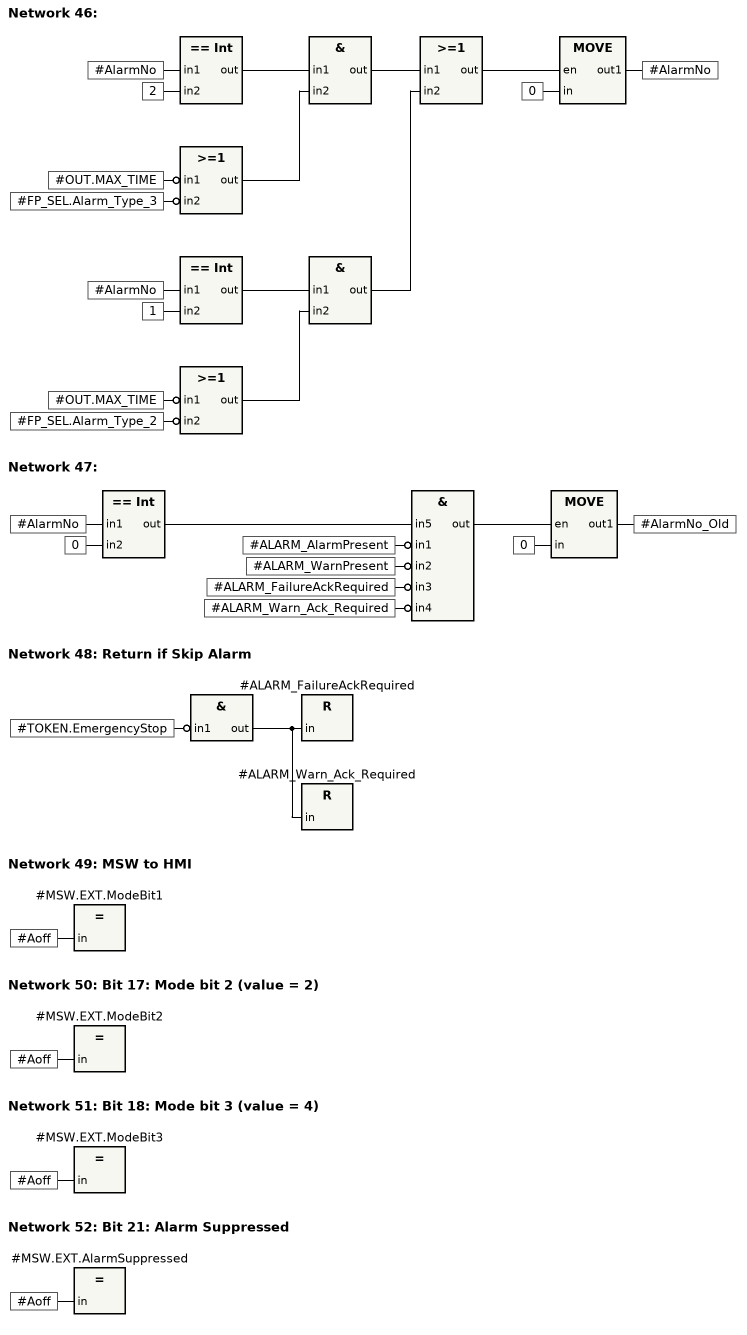
   IF ((#AlarmNo = 2) AND (NOT #OUT.MAX_TIME OR NOT #FP_SEL.Alarm_Type_3)) OR ((#AlarmNo = 1) AND (NOT #OUT.MAX_TIME OR NOT #FP_SEL.Alarm_Type_2)) THEN
       #AlarmNo := 0;
   END_IF;
END_REGION

REGION Network 47
   IF (#AlarmNo = 0) AND NOT #ALARM_AlarmPresent AND NOT #ALARM_WarnPresent AND NOT #ALARM_FailureAckRequired AND NOT #ALARM_Warn_Ack_Required THEN
       #AlarmNo_Old := 0;
   END_IF;
END_REGION

REGION Network 48: Return if Skip Alarm
   Skip:
   IF NOT #TOKEN.EmergencyStop THEN
       #ALARM_FailureAckRequired := FALSE;
       #ALARM_Warn_Ack_Required := FALSE;
   END_IF;
END_REGION

REGION Network 49: MSW to HMI
   #MSW.EXT.ModeBit1 := #Aoff;
END_REGION

REGION Network 50: Bit 17: Mode bit 2 (value = 2)
   #MSW.EXT.ModeBit2 := #Aoff;
END_REGION

REGION Network 51: Bit 18: Mode bit 3 (value = 4)
   #MSW.EXT.ModeBit3 := #Aoff;
END_REGION

REGION Network 52: Bit 21: Alarm Suppressed
   #MSW.EXT.AlarmSuppressed := #Aoff;
END_REGION

REGION Network 53: Bit 22: Alarm Condition Present
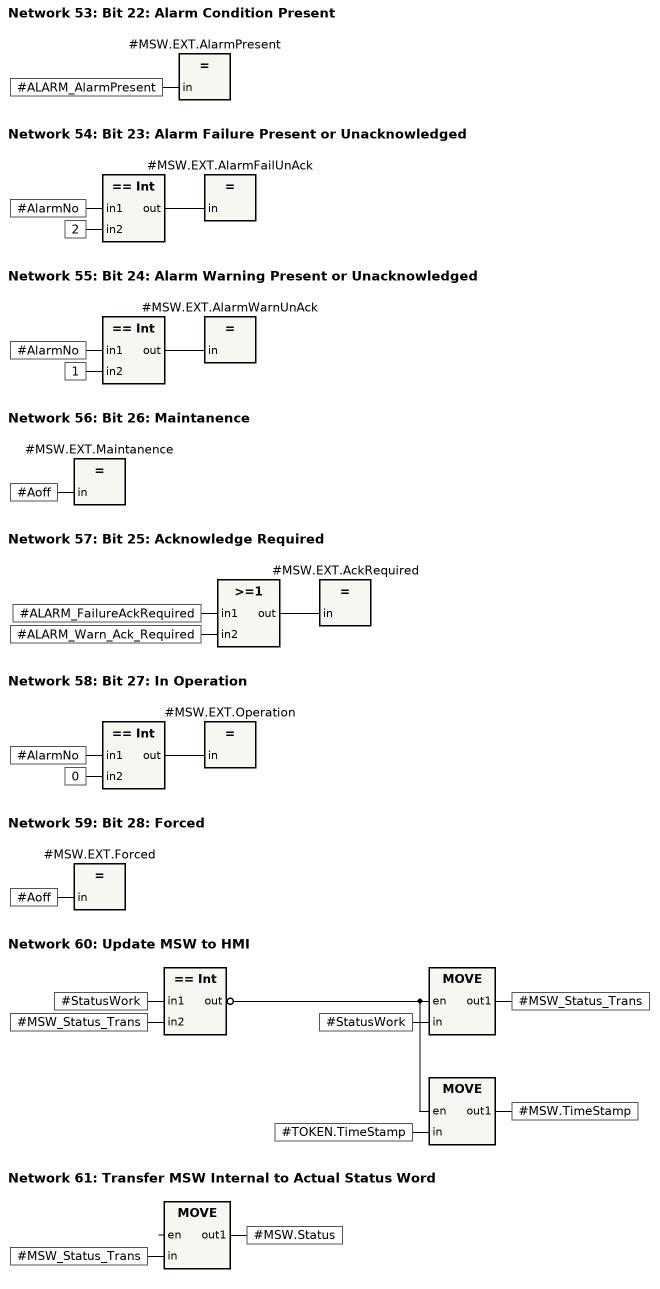
   #MSW.EXT.AlarmPresent := #ALARM_AlarmPresent;
END_REGION

REGION Network 54: Bit 23: Alarm Failure Present or Unacknowledged
   #MSW.EXT.AlarmFailUnAck := #AlarmNo = 2;
END_REGION

REGION Network 55: Bit 24: Alarm Warning Present or Unacknowledged
   #MSW.EXT.AlarmWarnUnAck := #AlarmNo = 1;
END_REGION

REGION Network 56: Bit 26: Maintanence
   #MSW.EXT.Maintanence := #Aoff;
END_REGION

REGION Network 57: Bit 25: Acknowledge Required
   #MSW.EXT.AckRequired := #ALARM_FailureAckRequired OR #ALARM_Warn_Ack_Required;
END_REGION

REGION Network 58: Bit 27: In Operation
   #MSW.EXT.Operation := #AlarmNo = 0;
END_REGION

REGION Network 59: Bit 28: Forced
   #MSW.EXT.Forced := #Aoff;
END_REGION

REGION Network 60: Update MSW to HMI
   #_w1 := NOT (#StatusWork = #MSW_Status_Trans);
   IF #_w1 THEN
       #MSW_Status_Trans := #StatusWork;
       #MSW.TimeStamp := #TOKEN.TimeStamp;
   END_IF;
END_REGION

REGION Network 61: Transfer MSW Internal to Actual Status Word
   #MSW.Status := #MSW_Status_Trans;
END_REGION

REGION Network 62: Write STAT to OUT
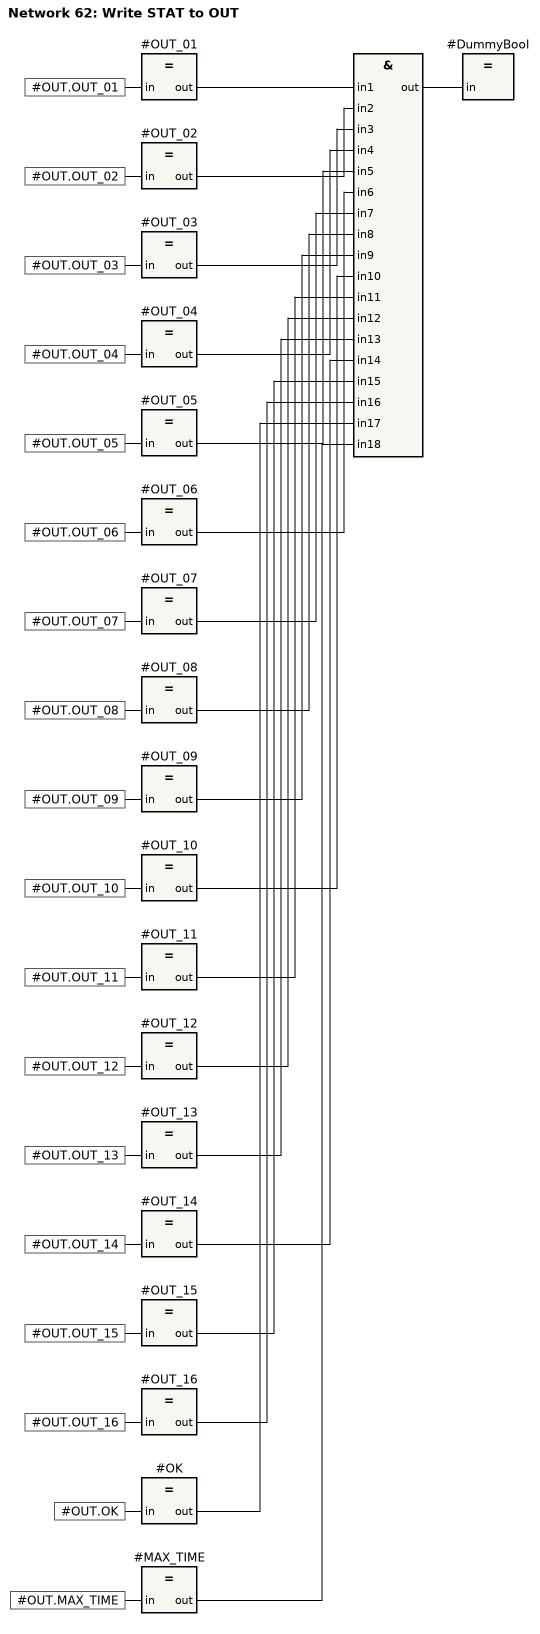
   #OUT_01 := #OUT.OUT_01;
   #OUT_02 := #OUT.OUT_02;
   #OUT_03 := #OUT.OUT_03;
   #OUT_04 := #OUT.OUT_04;
   #OUT_05 := #OUT.OUT_05;
   #OUT_06 := #OUT.OUT_06;
   #OUT_07 := #OUT.OUT_07;
   #OUT_08 := #OUT.OUT_08;
   #OUT_09 := #OUT.OUT_09;
   #OUT_10 := #OUT.OUT_10;
   #OUT_11 := #OUT.OUT_11;
   #OUT_12 := #OUT.OUT_12;
   #OUT_13 := #OUT.OUT_13;
   #OUT_14 := #OUT.OUT_14;
   #OUT_15 := #OUT.OUT_15;
   #OUT_16 := #OUT.OUT_16;
   #OK := #OUT.OK;
   #MAX_TIME := #OUT.MAX_TIME;
   #DummyBool := #OUT.OUT_01 AND #OUT.OUT_02 AND #OUT.OUT_03 AND #OUT.OUT_04 AND #OUT.OUT_05 AND #OUT.OUT_06 AND #OUT.OUT_07 AND #OUT.OUT_08 AND #OUT.OUT_09 AND #OUT.OUT_10 AND #OUT.OUT_11 AND #OUT.OUT_12 AND #OUT.OUT_13 AND #OUT.OUT_14 AND #OUT.OUT_15 AND #OUT.OUT_16 AND #OUT.OK AND #OUT.MAX_TIME;
END_REGION
END_FUNCTION_BLOCK

FUNCTION_BLOCK "ACESYS_ALTERNATE"   // FB232, FBD
TITLE = ACESYS V8.0 - Build 003 - ALTERNATE
{ S7_Optimized_Access := 'FALSE' }
AUTHOR : FLSmidth
FAMILY : ACESYS
NAME : ALTERNAT
VERSION : 8.0
// Structure of this FB:
// 
// The FB contain the following program sections:
// 
// 1) HourCounters
// 2) Priority arrangement for Auto sequence (sorting etc)
// 3) Sorting of manual priority
// 4) Detection of Load one more compressor
// 5) Detection of Unload one compressor
// 6) Detection of priority change by timer in Auto
// 7) Detect number of units running
// 8) Create final priority acording to selected mode
// 9) Create ASTR command
// 10) Avoid that more compressors start at the same time
// 11) Indication for priority change in progress
// 12) Set LOAD Commands
// 13) Indication Bar on faceplate
   VAR_INPUT
      PID_CV : Real;   // Output from PID
      Unit01_OK : Bool := TRUE;   // Unit 1 OK
      Unit01_SACK : Bool;   // Unit 1 Start Acknowledged
      Unit01_RD : Bool;   // Unit 1 Motor Run Delayed
      Unit02_OK : Bool := TRUE;   // Unit 2 OK
      Unit02_SACK : Bool;   // Unit 2 Start Acknowledged
      Unit02_RD : Bool;   // Unit 2 Motor Run Delayed
      Unit03_OK : Bool := TRUE;   // Unit 3 OK
      Unit03_SACK : Bool;   // Unit 3 Start Acknowledged
      Unit03_RD : Bool;   // Unit 3 Motor Run Delayed
      Unit04_OK : Bool := TRUE;   // Unit 4 OK
      Unit04_SACK : Bool;   // Unit 4 Start Acknowledged
      Unit04_RD : Bool;   // Unit 4 Motor Run Delayed
      Unit05_OK : Bool := TRUE;   // Unit 5 OK
      Unit05_SACK : Bool;   // Unit 5 Start Acknowledged
      Unit05_RD : Bool;   // Unit 5 Motor Run Delayed
      Unit06_OK : Bool := TRUE;   // Unit 6 OK
      Unit06_SACK : Bool;   // Unit 6 Start Acknowledged
      Unit06_RD : Bool;   // Unit 6 Motor Run Delayed
      Unit07_OK : Bool := TRUE;   // Unit 7 OK
      Unit07_SACK : Bool;   // Unit 7 Start Acknowledged
      Unit07_RD : Bool;   // Unit 7 Motor Run Delayed
      Unit08_OK : Bool := TRUE;   // Unit 8 OK
      Unit08_SACK : Bool;   // Unit 8 Start Acknowledged
      Unit08_RD : Bool;   // Unit 8 Motor Run Delayed
      Unit09_OK : Bool := TRUE;   // Unit 9 OK
      Unit09_SACK : Bool;   // Unit 9 Start Acknowledged
      Unit09_RD : Bool;   // Unit 9 Motor Run Delayed
      Unit10_OK : Bool := TRUE;   // Unit 10 OK
      Unit10_SACK : Bool;   // Unit 10 Start Acknowledged
      Unit10_RD : Bool;   // Unit 10 Motor Run Delayed
   END_VAR
   VAR_OUTPUT
      Unit01_LOAD : Bool;   // Unit 1 Load
      Unit01_SEL : Bool;   // Unit 1 Selected
      Unit01_ASTR : Bool;   // Unit 1 Auto Start
      Unit02_LOAD : Bool;   // Unit 2 Load
      Unit02_SEL : Bool;   // Unit 2 Selected
      Unit02_ASTR : Bool;   // Unit 2 Auto Start
      Unit03_LOAD : Bool;   // Unit 3 Load
      Unit03_SEL : Bool;   // Unit 3 Selected
      Unit03_ASTR : Bool;   // Unit 3 Auto Start
      Unit04_LOAD : Bool;   // Unit 4 Load
      Unit04_SEL : Bool;   // Unit 4 Selected
      Unit04_ASTR : Bool;   // Unit 4 Auto Start
      Unit05_LOAD : Bool;   // Unit 5 Load
      Unit05_SEL : Bool;   // Unit 5 Selected
      Unit05_ASTR : Bool;   // Unit 5 Auto Start
      Unit06_LOAD : Bool;   // Unit 6 Load
      Unit06_SEL : Bool;   // Unit 6 Selected
      Unit06_ASTR : Bool;   // Unit 6 Auto Start
      Unit07_LOAD : Bool;   // Unit 7 Load
      Unit07_SEL : Bool;   // Unit 7 Selected
      Unit07_ASTR : Bool;   // Unit 7 Auto Start
      Unit08_LOAD : Bool;   // Unit 8 Load
      Unit08_SEL : Bool;   // Unit 8 Selected
      Unit08_ASTR : Bool;   // Unit 8 Auto Start
      Unit09_LOAD : Bool;   // Unit 9 Load
      Unit09_SEL : Bool;   // Unit 9 Selected
      Unit09_ASTR : Bool;   // Unit 9 Auto Start
      Unit10_LOAD : Bool;   // Unit 10 Load
      Unit10_SEL : Bool;   // Unit 10 Selected
      Unit10_ASTR : Bool;   // Unit 10 Auto Start
      MSW : "ACESYS_HMI_STAT_32T";
   END_VAR
   VAR_IN_OUT
      TOKEN : "ACESYS_TOKEN";
   END_VAR
   VAR
      BlockInfo : Struct
         Ace_Version : Int;   // Acesys Block Version Number
         Ace_BuildNo : Int;   // Acesys Block Build Number
         DB_Number : Int;   // Block Instance DB Number
      END_STRUCT;
      FP_CMD : Struct   // Faceplate Commands
         Spare_08 : Bool;
         Spare_09 : Bool;
         Spare_10 : Bool;
         Spare_11 : Bool;
         Spare_12 : Bool;
         Spare_13 : Bool;
         Spare_14 : Bool;
         AckAlarm : Bool;   // Alarm Acknowledge
         Spare_00 : Bool;
         Spare_01 : Bool;
         Spare_02 : Bool;
         Spare_03 : Bool;
         Spare_04 : Bool;
         Spare_05 : Bool;
         Spare_06 : Bool;
         Spare_07 : Bool;
      END_STRUCT;
      FP_PARM : Struct
         NoOfUnits : Int := 6;   // Number of Units to be controlled
         NoToRun : Int;   // Number of Units that shall run
         RunTime_Unit01 : Real;
         RunTime_Unit02 : Real;
         RunTime_Unit03 : Real;
         RunTime_Unit04 : Real;
         RunTime_Unit05 : Real;
         RunTime_Unit06 : Real;
         RunTime_Unit07 : Real;
         RunTime_Unit08 : Real;
         RunTime_Unit09 : Real;
         RunTime_Unit10 : Real;
         ManPrio_Unit01 : Int := 1;
         ManPrio_Unit02 : Int := 2;
         ManPrio_Unit03 : Int := 3;
         ManPrio_Unit04 : Int := 4;
         ManPrio_Unit05 : Int := 5;
         ManPrio_Unit06 : Int := 6;
         ManPrio_Unit07 : Int := 7;
         ManPrio_Unit08 : Int := 8;
         ManPrio_Unit09 : Int := 9;
         ManPrio_Unit10 : Int := 10;
         IncDelay_Pre : Int := 10;
         IncDelay_ACC : Int;
         DecDelay_Pre : Int := 10;
         Dec_Delay_ACC : Int;
         ShiftTime_PRE : Int := 60;
         ShiftTime_ACC : Int;
         SelectivityTime_PRE : Int := 5;
         SelectivityTime_ACC : Int;
         Delayed_RD_PRE : Int;
      END_STRUCT;
      FP_PrioFinal : Array[1..10] of Int;   // Active Priority (Sorted)
      FP_PrioMan : Array[1..10] of Int;   // Manual Priority (Sorted)
      FP_PrioAuto : Array[1..10] of Int;   // Auto Priority (Sorted)
      FP_SEL : Struct
         Seq_Auto : Bool;
         Seq_Manual : Bool;
         Load : Bool;
         Unit01_SEL : Bool;
         Unit02_SEL : Bool;
         Unit03_SEL : Bool;
         Unit04_SEL : Bool;
         Unit05_SEL : Bool;
         Unit06_SEL : Bool;
         Unit07_SEL : Bool;
         Unit08_SEL : Bool;
         Unit09_SEL : Bool;
         Unit10_SEL : Bool;
         Spare03 : Bool;
         Spare02 : Bool;
         Spare01 : Bool;
      END_STRUCT;
      ONS : Struct
         Seq_Auto_On : Bool;
         Seq_Manual_On : Bool;
         Seq_Auto_Off : Bool;
         Seq_Manual_Off : Bool;
         Seq_Auto : Bool;
         PriorityProgress : Bool;
         Spare10 : Bool;
         Spare09 : Bool;
         Spare08 : Bool;
         Spare07 : Bool;
         Spare06 : Bool;
         Spare05 : Bool;
         Spare04 : Bool;
         Spare03 : Bool;
         Spare02 : Bool;
         Spare01 : Bool;
      END_STRUCT;
      StatusWork : Int;
      A_Prio_Hours : Array[1..10] of DInt;
      MPN : Array[1..10] of Int;
      IncDelay_Mem : Int;
      DecDelay_Mem : Int;
      SelectivityTime_MEM : Int;
      Old_Sxx : Int;   // Old Sxx
      Act_Sxx : Int;
      Act_Sxx_AT AT Act_Sxx : Array[1..16] of Bool;
      UnitsRunning : Int;   // Hold the number of running Units
      Unit01_Delayed_RD_Mem : Int;
      Unit02_Delayed_RD_Mem : Int;
      Unit03_Delayed_RD_Mem : Int;
      Unit04_Delayed_RD_Mem : Int;
      Unit05_Delayed_RD_Mem : Int;
      Unit06_Delayed_RD_Mem : Int;
      Unit07_Delayed_RD_Mem : Int;
      Unit08_Delayed_RD_Mem : Int;
      Unit09_Delayed_RD_Mem : Int;
      Unit10_Delayed_RD_Mem : Int;
      INC : Bool;   // Increace Number of Unites
      DEC : Bool;   // Decreace Number of Unites
      ChangePriority : Bool;
      WaitForRD : Bool;
      PriorityProgress : Bool;
      PriorityChange : Bool;   // Priority Change in Progress
      Unit01_CMD : Bool;   // Intermidiate command 1
      Unit02_CMD : Bool;   // Intermidiate command 2
      Unit03_CMD : Bool;   // Intermidiate command 3
      Unit04_CMD : Bool;   // Intermidiate command 4
      Unit05_CMD : Bool;   // Intermidiate command 5
      Unit06_CMD : Bool;   // Intermidiate command 6
      Unit07_CMD : Bool;   // Intermidiate command 7
      Unit08_CMD : Bool;   // Intermidiate command 8
      Unit09_CMD : Bool;   // Intermidiate command 9
      Unit10_CMD : Bool;   // Intermidiate command 10
      Unit01_Act_CMD : Bool;   // Unit 1: Active Command
      Unit02_Act_CMD : Bool;   // Unit 2: Active Command
      Unit03_Act_CMD : Bool;   // Unit 3: Active Command
      Unit04_Act_CMD : Bool;   // Unit 4: Active Command
      Unit05_Act_CMD : Bool;   // Unit 5: Active Command
      Unit06_Act_CMD : Bool;   // Unit 6: Active Command
      Unit07_Act_CMD : Bool;   // Unit 7: Active Command
      Unit08_Act_CMD : Bool;   // Unit 8: Active Command
      Unit09_Act_CMD : Bool;   // Unit 9: Active Command
      Unit10_Act_CMD : Bool;   // Unit 10: Active Command
      SpareBool_06 : Bool;
      SpareBool_05 : Bool;
      SpareBool_04 : Bool;
      SpareBool_03 : Bool;
      SpareBool_02 : Bool;
      SpareBool_01 : Bool;
      OUT : Struct
         Unit01_LOAD : Bool;
         Unit01_SEL : Bool;
         Unit01_ASTR : Bool;
         Unit02_LOAD : Bool;
         Unit02_SEL : Bool;
         Unit02_ASTR : Bool;
         Unit03_LOAD : Bool;
         Unit03_SEL : Bool;
         Unit03_ASTR : Bool;
         Unit04_LOAD : Bool;
         Unit04_SEL : Bool;
         Unit04_ASTR : Bool;
         Unit05_LOAD : Bool;
         Unit05_SEL : Bool;
         Unit05_ASTR : Bool;
         Unit06_LOAD : Bool;
         Unit06_SEL : Bool;
         Unit06_ASTR : Bool;
         Unit07_LOAD : Bool;
         Unit07_SEL : Bool;
         Unit07_ASTR : Bool;
         Unit08_LOAD : Bool;
         Unit08_SEL : Bool;
         Unit08_ASTR : Bool;
         Unit09_LOAD : Bool;
         Unit09_SEL : Bool;
         Unit09_ASTR : Bool;
         Unit10_LOAD : Bool;
         Unit10_SEL : Bool;
         Unit10_ASTR : Bool;
      END_STRUCT;
      MSW_Status_Trans : Int;
   END_VAR
   VAR_TEMP
      Unit01_RDY : Bool;
      Unit02_RDY : Bool;
      Unit03_RDY : Bool;
      Unit04_RDY : Bool;
      Unit05_RDY : Bool;
      Unit06_RDY : Bool;
      Unit07_RDY : Bool;
      Unit08_RDY : Bool;
      Unit09_RDY : Bool;
      Unit10_RDY : Bool;
      Unit11_Spare : Bool;
      Unit12_Spare : Bool;
      Unit13_Spare : Bool;
      Unit14_Spare : Bool;
      Unit15_Spare : Bool;
      Unit16_Spare : Bool;
      Aon : Bool;
      Aoff : Bool;
      DummyBool : Bool;
      SortChange : Bool;
      SelectivityTime_Done : Bool;
      Delayed_RD_Done : Bool;
      TempDINT : DInt;
      TempREAL : Real;
      TempINT : Int;
      SaveAR1 : DWord;
      SaveAR2 : DWord;
      TempH01 : Real;
      TempH02 : Real;
      TempH03 : Real;
      TempH04 : Real;
      TempH05 : Real;
      TempH06 : Real;
      TempH07 : Real;
      TempH08 : Real;
      TempH09 : Real;
      TempH10 : Real;
      TempP01 : Int;
      TempP02 : Int;
      TempP03 : Int;
      TempP04 : Int;
      TempP05 : Int;
      TempP06 : Int;
      TempP07 : Int;
      TempP08 : Int;
      TempP09 : Int;
      TempP10 : Int;
      UnitCount : Int;   // Number of Units selected
      SortCounter : Int;   // Counter used in bubbel sort
      MaxUnitsReady : Int;
      PID_NoOfCom_SP : Int;
      Temp_CMD : Int;
      RunLoop : Int;
      OFFSET : Int;
      "OFFSET+1" : Int;
   END_VAR
   VAR_TEMP   // added for the SCL form of the ladder/FBD networks
      _w1 : Bool;
      _w2 : Bool;
      _w3 : Bool;
      _w4 : Bool;
      _w5 : Bool;
      _w6 : Bool;
      _w7 : Bool;
      _w8 : Bool;
      _w9 : Bool;
      _w10 : Bool;
   END_VAR
BEGIN

REGION Network 1
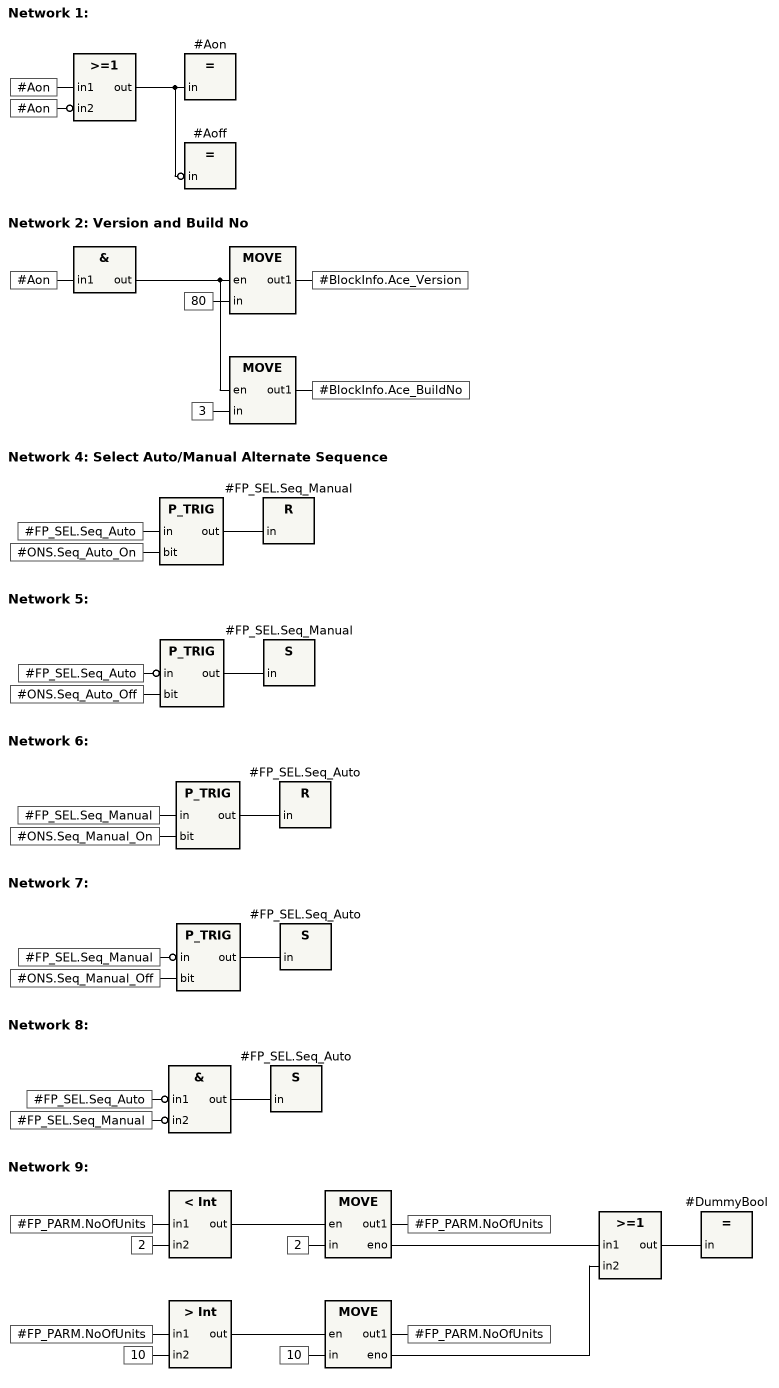
   #Aon := #Aon OR NOT #Aon;
   #Aoff := NOT #Aon;
END_REGION

REGION Network 2: Version and Build No
   IF #Aon THEN
       #BlockInfo.Ace_Version := 80;
       #BlockInfo.Ace_BuildNo := 3;
   END_IF;
END_REGION

REGION Network 3 (STL): Instance DB Number to Faceplate
         L     DINO;
         T     #BlockInfo.DB_Number;
END_REGION

REGION Network 4: Select Auto/Manual Alternate Sequence
   #_w1 := #FP_SEL.Seq_Auto AND NOT #ONS.Seq_Auto_On;   // rising edge
   #ONS.Seq_Auto_On := #FP_SEL.Seq_Auto;
   IF #_w1 THEN #FP_SEL.Seq_Manual := FALSE; END_IF;
END_REGION

REGION Network 5
   #_w1 := NOT #FP_SEL.Seq_Auto AND NOT #ONS.Seq_Auto_Off;   // rising edge
   #ONS.Seq_Auto_Off := NOT #FP_SEL.Seq_Auto;
   IF #_w1 THEN #FP_SEL.Seq_Manual := TRUE; END_IF;
END_REGION

REGION Network 6
   #_w1 := #FP_SEL.Seq_Manual AND NOT #ONS.Seq_Manual_On;   // rising edge
   #ONS.Seq_Manual_On := #FP_SEL.Seq_Manual;
   IF #_w1 THEN #FP_SEL.Seq_Auto := FALSE; END_IF;
END_REGION

REGION Network 7
   #_w1 := NOT #FP_SEL.Seq_Manual AND NOT #ONS.Seq_Manual_Off;   // rising edge
   #ONS.Seq_Manual_Off := NOT #FP_SEL.Seq_Manual;
   IF #_w1 THEN #FP_SEL.Seq_Auto := TRUE; END_IF;
END_REGION

REGION Network 8
   IF NOT #FP_SEL.Seq_Auto AND NOT #FP_SEL.Seq_Manual THEN #FP_SEL.Seq_Auto := TRUE; END_IF;
END_REGION

REGION Network 9
   // ENO of a box is taken as its EN; it also drops when the box reports an error
   #_w1 := #FP_PARM.NoOfUnits < 2;
   IF #_w1 THEN #FP_PARM.NoOfUnits := 2; END_IF;
   #_w2 := #FP_PARM.NoOfUnits > 10;
   IF #_w2 THEN #FP_PARM.NoOfUnits := 10; END_IF;
   #DummyBool := #_w1 OR #_w2;
END_REGION

REGION Network 10
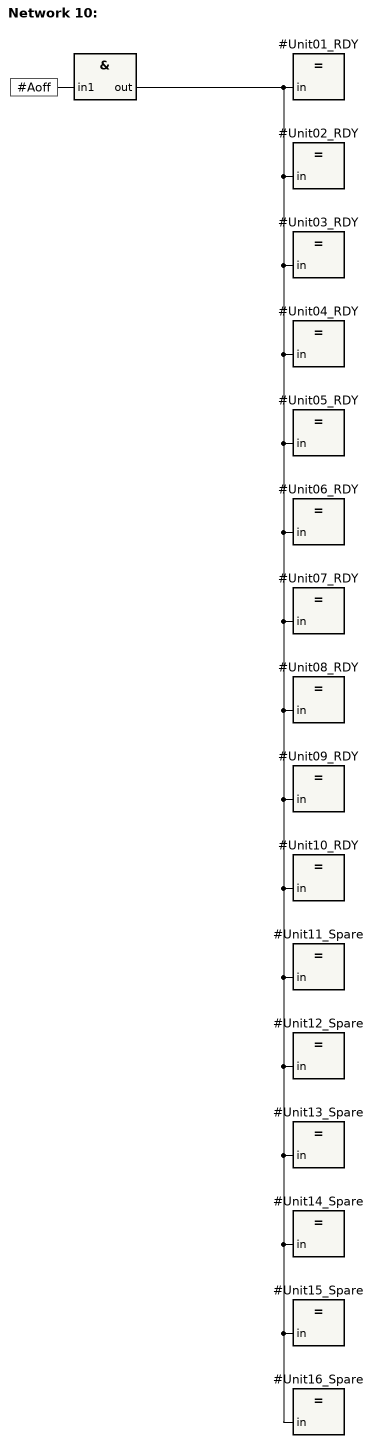
   #Unit01_RDY := #Aoff;
   #Unit02_RDY := #Aoff;
   #Unit03_RDY := #Aoff;
   #Unit04_RDY := #Aoff;
   #Unit05_RDY := #Aoff;
   #Unit06_RDY := #Aoff;
   #Unit07_RDY := #Aoff;
   #Unit08_RDY := #Aoff;
   #Unit09_RDY := #Aoff;
   #Unit10_RDY := #Aoff;
   #Unit11_Spare := #Aoff;
   #Unit12_Spare := #Aoff;
   #Unit13_Spare := #Aoff;
   #Unit14_Spare := #Aoff;
   #Unit15_Spare := #Aoff;
   #Unit16_Spare := #Aoff;
END_REGION

REGION Network 11: Set flags for Selected, OK and SACK
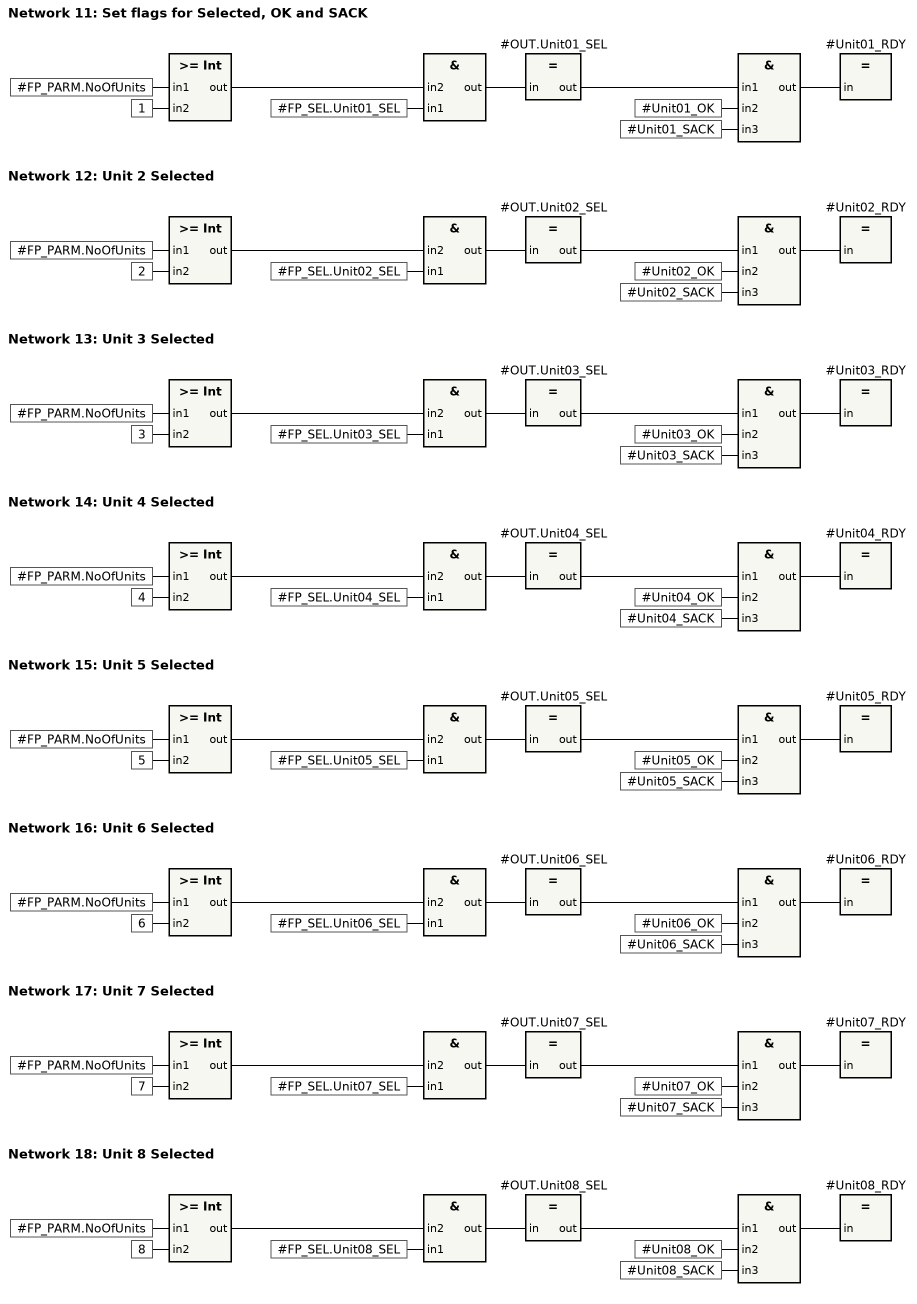
   #OUT.Unit01_SEL := (#FP_PARM.NoOfUnits >= 1) AND #FP_SEL.Unit01_SEL;
   #Unit01_RDY := #OUT.Unit01_SEL AND #Unit01_OK AND #Unit01_SACK;
END_REGION

REGION Network 12: Unit 2 Selected
   #OUT.Unit02_SEL := (#FP_PARM.NoOfUnits >= 2) AND #FP_SEL.Unit02_SEL;
   #Unit02_RDY := #OUT.Unit02_SEL AND #Unit02_OK AND #Unit02_SACK;
END_REGION

REGION Network 13: Unit 3 Selected
   #OUT.Unit03_SEL := (#FP_PARM.NoOfUnits >= 3) AND #FP_SEL.Unit03_SEL;
   #Unit03_RDY := #OUT.Unit03_SEL AND #Unit03_OK AND #Unit03_SACK;
END_REGION

REGION Network 14: Unit 4 Selected
   #OUT.Unit04_SEL := (#FP_PARM.NoOfUnits >= 4) AND #FP_SEL.Unit04_SEL;
   #Unit04_RDY := #OUT.Unit04_SEL AND #Unit04_OK AND #Unit04_SACK;
END_REGION

REGION Network 15: Unit 5 Selected
   #OUT.Unit05_SEL := (#FP_PARM.NoOfUnits >= 5) AND #FP_SEL.Unit05_SEL;
   #Unit05_RDY := #OUT.Unit05_SEL AND #Unit05_OK AND #Unit05_SACK;
END_REGION

REGION Network 16: Unit 6 Selected
   #OUT.Unit06_SEL := (#FP_PARM.NoOfUnits >= 6) AND #FP_SEL.Unit06_SEL;
   #Unit06_RDY := #OUT.Unit06_SEL AND #Unit06_OK AND #Unit06_SACK;
END_REGION

REGION Network 17: Unit 7 Selected
   #OUT.Unit07_SEL := (#FP_PARM.NoOfUnits >= 7) AND #FP_SEL.Unit07_SEL;
   #Unit07_RDY := #OUT.Unit07_SEL AND #Unit07_OK AND #Unit07_SACK;
END_REGION

REGION Network 18: Unit 8 Selected
   #OUT.Unit08_SEL := (#FP_PARM.NoOfUnits >= 8) AND #FP_SEL.Unit08_SEL;
   #Unit08_RDY := #OUT.Unit08_SEL AND #Unit08_OK AND #Unit08_SACK;
END_REGION

REGION Network 19: Unit 9 Selected
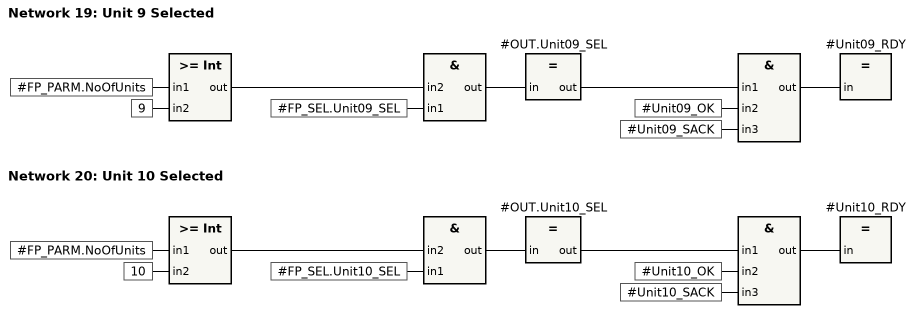
   #OUT.Unit09_SEL := (#FP_PARM.NoOfUnits >= 9) AND #FP_SEL.Unit09_SEL;
   #Unit09_RDY := #OUT.Unit09_SEL AND #Unit09_OK AND #Unit09_SACK;
END_REGION

REGION Network 20: Unit 10 Selected
   #OUT.Unit10_SEL := (#FP_PARM.NoOfUnits >= 10) AND #FP_SEL.Unit10_SEL;
   #Unit10_RDY := #OUT.Unit10_SEL AND #Unit10_OK AND #Unit10_SACK;
END_REGION

REGION Network 21: Save the actual select status
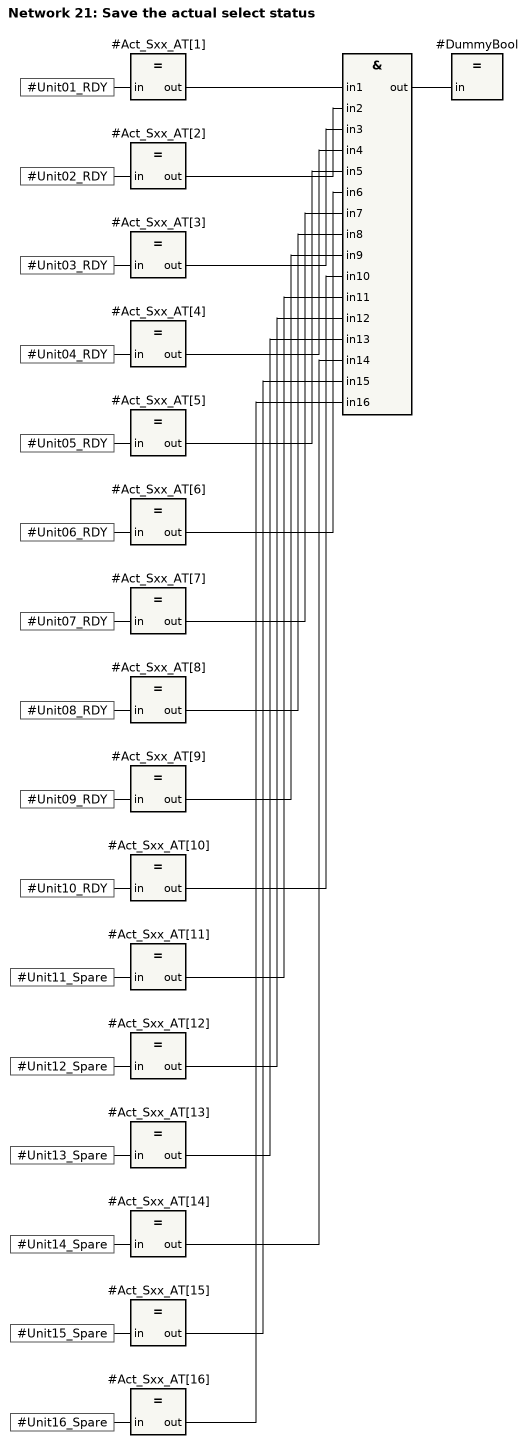
   #Act_Sxx_AT[1] := #Unit01_RDY;
   #Act_Sxx_AT[2] := #Unit02_RDY;
   #Act_Sxx_AT[3] := #Unit03_RDY;
   #Act_Sxx_AT[4] := #Unit04_RDY;
   #Act_Sxx_AT[5] := #Unit05_RDY;
   #Act_Sxx_AT[6] := #Unit06_RDY;
   #Act_Sxx_AT[7] := #Unit07_RDY;
   #Act_Sxx_AT[8] := #Unit08_RDY;
   #Act_Sxx_AT[9] := #Unit09_RDY;
   #Act_Sxx_AT[10] := #Unit10_RDY;
   #Act_Sxx_AT[11] := #Unit11_Spare;
   #Act_Sxx_AT[12] := #Unit12_Spare;
   #Act_Sxx_AT[13] := #Unit13_Spare;
   #Act_Sxx_AT[14] := #Unit14_Spare;
   #Act_Sxx_AT[15] := #Unit15_Spare;
   #Act_Sxx_AT[16] := #Unit16_Spare;
   #DummyBool := #Unit01_RDY AND #Unit02_RDY AND #Unit03_RDY AND #Unit04_RDY AND #Unit05_RDY AND #Unit06_RDY AND #Unit07_RDY AND #Unit08_RDY AND #Unit09_RDY AND #Unit10_RDY AND #Unit11_Spare AND #Unit12_Spare AND #Unit13_Spare AND #Unit14_Spare AND #Unit15_Spare AND #Unit16_Spare;
END_REGION

REGION Network 22
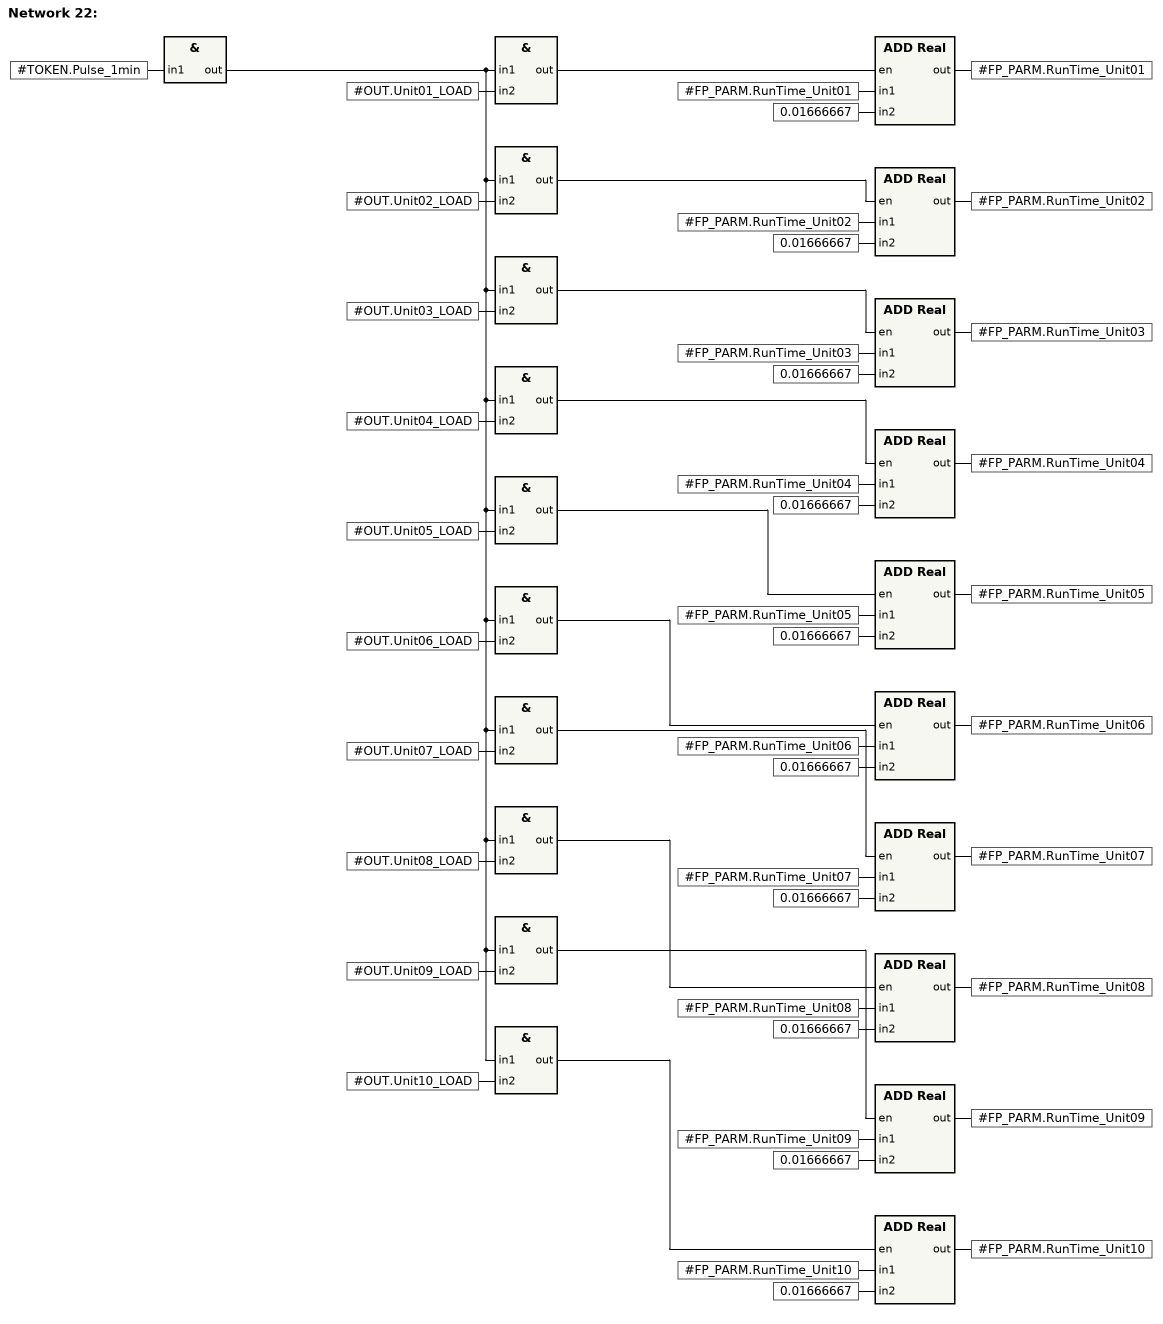
   IF #TOKEN.Pulse_1min AND #OUT.Unit01_LOAD THEN
       #FP_PARM.RunTime_Unit01 := #FP_PARM.RunTime_Unit01 + 0.01666667;
   END_IF;
   IF #TOKEN.Pulse_1min AND #OUT.Unit02_LOAD THEN
       #FP_PARM.RunTime_Unit02 := #FP_PARM.RunTime_Unit02 + 0.01666667;
   END_IF;
   IF #TOKEN.Pulse_1min AND #OUT.Unit03_LOAD THEN
       #FP_PARM.RunTime_Unit03 := #FP_PARM.RunTime_Unit03 + 0.01666667;
   END_IF;
   IF #TOKEN.Pulse_1min AND #OUT.Unit04_LOAD THEN
       #FP_PARM.RunTime_Unit04 := #FP_PARM.RunTime_Unit04 + 0.01666667;
   END_IF;
   IF #TOKEN.Pulse_1min AND #OUT.Unit05_LOAD THEN
       #FP_PARM.RunTime_Unit05 := #FP_PARM.RunTime_Unit05 + 0.01666667;
   END_IF;
   IF #TOKEN.Pulse_1min AND #OUT.Unit06_LOAD THEN
       #FP_PARM.RunTime_Unit06 := #FP_PARM.RunTime_Unit06 + 0.01666667;
   END_IF;
   IF #TOKEN.Pulse_1min AND #OUT.Unit07_LOAD THEN
       #FP_PARM.RunTime_Unit07 := #FP_PARM.RunTime_Unit07 + 0.01666667;
   END_IF;
   IF #TOKEN.Pulse_1min AND #OUT.Unit08_LOAD THEN
       #FP_PARM.RunTime_Unit08 := #FP_PARM.RunTime_Unit08 + 0.01666667;
   END_IF;
   IF #TOKEN.Pulse_1min AND #OUT.Unit09_LOAD THEN
       #FP_PARM.RunTime_Unit09 := #FP_PARM.RunTime_Unit09 + 0.01666667;
   END_IF;
   IF #TOKEN.Pulse_1min AND #OUT.Unit10_LOAD THEN
       #FP_PARM.RunTime_Unit10 := #FP_PARM.RunTime_Unit10 + 0.01666667;
   END_IF;
END_REGION

REGION Network 23: 2) Priority arrangement for Auto sequence
   // Create temp vars.
   // Because using AR1 and AR2 inhibits use of block parameters between the load of 
   // the pointer and the use of it, the selects are copied to internal variables
   // (This is because the FB also uses the AR1 and AR2 to access the block 
   // parameters
   // 
   // Copy selects to temp.vars
   // Copy hours to temp.vars
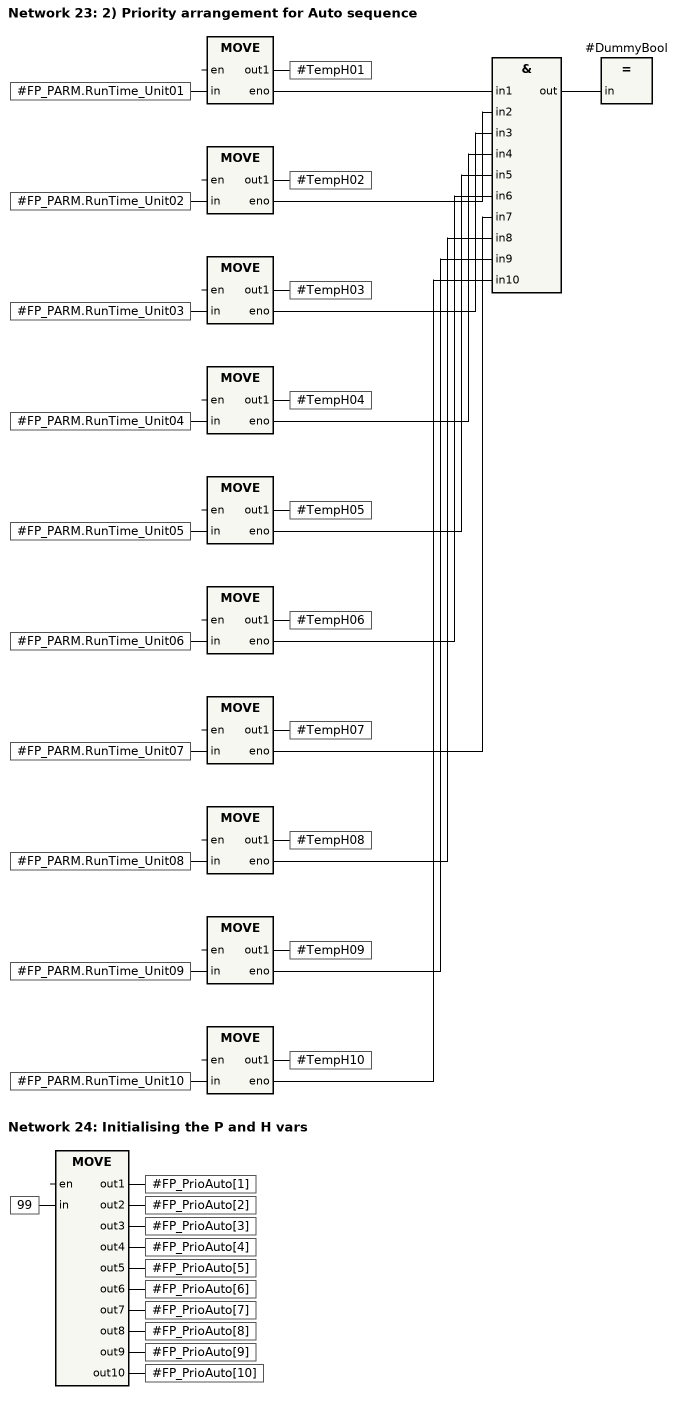
   #TempH01 := #FP_PARM.RunTime_Unit01;
   #TempH02 := #FP_PARM.RunTime_Unit02;
   #TempH03 := #FP_PARM.RunTime_Unit03;
   #TempH04 := #FP_PARM.RunTime_Unit04;
   #TempH05 := #FP_PARM.RunTime_Unit05;
   #TempH06 := #FP_PARM.RunTime_Unit06;
   #TempH07 := #FP_PARM.RunTime_Unit07;
   #TempH08 := #FP_PARM.RunTime_Unit08;
   #TempH09 := #FP_PARM.RunTime_Unit09;
   #TempH10 := #FP_PARM.RunTime_Unit10;
   #DummyBool := TRUE;
END_REGION

REGION Network 24: Initialising the P and H vars
   #FP_PrioAuto[1] := 99;
   #FP_PrioAuto[2] := 99;
   #FP_PrioAuto[3] := 99;
   #FP_PrioAuto[4] := 99;
   #FP_PrioAuto[5] := 99;
   #FP_PrioAuto[6] := 99;
   #FP_PrioAuto[7] := 99;
   #FP_PrioAuto[8] := 99;
   #FP_PrioAuto[9] := 99;
   #FP_PrioAuto[10] := 99;
END_REGION

REGION Network 25: Initialising the P and H vars
